C07140=1014.541,221.551,-132.905,168.191,53.842,160.168
C07141=1014.536,221.303,-132.880,168.186,53.852,160.169
C07142=1014.530,221.054,-132.855,168.181,53.862,160.170
C07143=1014.525,220.805,-132.830,168.177,53.871,160.171
C07144=1014.520,220.557,-132.805,168.172,53.881,160.172
C07145=1014.514,220.308,-132.780,168.167,53.891,160.173
C07146=1014.509,220.059,-132.754,168.163,53.900,160.174
C07147=1014.504,219.812,-132.730,168.159,53.910,160.176
C07148=1014.499,219.565,-132.705,168.154,53.919,160.177
C07149=1014.494,219.318,-132.680,168.149,53.929,160.178
C07150=1014.489,219.071,-132.655,168.144,53.939,160.179
C07151=1014.484,218.824,-132.630,168.140,53.948,160.180
C07152=1014.478,218.577,-132.606,168.136,53.959,160.181
C07153=1014.473,218.330,-132.581,168.131,53.969,160.182
C07154=1014.468,218.084,-132.556,168.126,53.978,160.183
C07155=1014.463,217.835,-132.531,168.123,53.988,160.185
C07156=1014.457,217.585,-132.507,168.118,53.997,160.186
C07157=1014.452,217.337,-132.482,168.113,54.008,160.187
C07158=1014.447,217.088,-132.457,168.109,54.018,160.188
C07159=1014.442,216.840,-132.433,168.104,54.027,160.189
C07160=1014.436,216.591,-132.408,168.099,54.038,160.190
C07161=1014.431,216.342,-132.384,168.095,54.048,160.191
C07162=1014.425,216.094,-132.359,168.090,54.058,160.193
C07163=1014.420,215.845,-132.334,168.085,54.068,160.194
C07164=1014.414,215.596,-132.309,168.081,54.078,160.195
C07165=1014.409,215.347,-132.285,168.076,54.088,160.196
C07166=1014.404,215.099,-132.261,168.072,54.099,160.198
C07167=1014.399,214.850,-132.236,168.067,54.108,160.199
C07168=1014.393,214.601,-132.211,168.063,54.119,160.200
C07169=1014.388,214.352,-132.187,168.058,54.129,160.201
C07170=1014.382,214.104,-132.162,168.054,54.139,160.202
C07171=1014.377,213.855,-132.138,168.049,54.149,160.203
C07172=1014.373,213.606,-132.113,168.045,54.159,160.205
C07173=1014.367,213.357,-132.088,168.040,54.169,160.206
C07174=1014.361,213.109,-132.064,168.035,54.180,160.207
C07175=1014.356,212.860,-132.040,168.031,54.190,160.208
C07176=1014.352,212.611,-132.015,168.026,54.200,160.209
C07177=1014.346,212.363,-131.991,168.022,54.211,160.211
C07178=1014.341,212.114,-131.966,168.017,54.220,160.212
C07179=1014.336,211.865,-131.942,168.013,54.231,160.213
C07180=1014.331,211.616,-131.917,168.008,54.241,160.214
C07181=1014.325,211.367,-131.893,168.004,54.251,160.215
C07182=1014.320,211.119,-131.868,168.000,54.262,160.217
C07183=1014.315,210.870,-131.844,167.995,54.272,160.218
C07184=1014.309,210.621,-131.820,167.991,54.282,160.219
C07185=1014.305,210.372,-131.795,167.986,54.293,160.220
C07186=1014.300,210.123,-131.772,167.982,54.303,160.222
C07187=1014.294,209.875,-131.747,167.977,54.313,160.223
C07188=1014.289,209.626,-131.723,167.973,54.324,160.224
C07189=1014.284,209.378,-131.699,167.969,54.334,160.226
C07190=1014.279,209.129,-131.675,167.963,54.345,160.227
C07191=1014.274,208.880,-131.650,167.959,54.355,160.228
C07192=1014.268,208.631,-131.625,167.954,54.365,160.229
C07193=1014.263,208.382,-131.601,167.950,54.376,160.230
C07194=1014.258,208.133,-131.577,167.946,54.386,160.232
C07195=1014.253,207.884,-131.553,167.942,54.397,160.233
C07196=1014.248,207.635,-131.529,167.936,54.408,160.234
C07197=1014.242,207.387,-131.505,167.932,54.418,160.236
C07198=1014.237,207.138,-131.481,167.928,54.429,160.237
C07199=1014.232,206.889,-131.457,167.924,54.440,160.238
C07200=1014.227,206.640,-131.433,167.919,54.450,160.239
C07201=1014.221,206.392,-131.409,167.914,54.461,160.241
C07202=1014.215,206.143,-131.385,167.910,54.472,160.242
C07203=1014.210,205.894,-131.362,167.906,54.482,160.243
C07204=1014.205,205.646,-131.337,167.901,54.493,160.245
C07205=1014.200,205.396,-131.314,167.896,54.504,160.246
C07206=1014.195,205.148,-131.290,167.892,54.514,160.247
C07207=1014.190,204.913,-131.267,167.887,54.524,160.248
C07208=1014.185,204.677,-131.245,167.884,54.534,160.250
C07209=1014.180,204.443,-131.222,167.880,54.545,160.251
C07210=1014.175,204.207,-131.200,167.875,54.555,160.252
C07211=1014.171,203.972,-131.178,167.871,54.565,160.253
C07212=1014.166,203.737,-131.155,167.866,54.575,160.254
C07213=1014.161,203.502,-131.133,167.863,54.585,160.256
C07214=1014.156,203.267,-131.110,167.859,54.596,160.257
C07215=1014.137,202.159,-131.012,167.332,54.506,160.118
C07216=1014.133,201.910,-130.990,167.327,54.518,160.120
C07217=1014.128,201.662,-130.968,167.321,54.530,160.121
C07218=1014.124,201.412,-130.946,167.316,54.542,160.122
C07219=1014.120,201.163,-130.924,167.312,54.554,160.124
C07220=1014.116,200.914,-130.902,167.307,54.566,160.125
C07221=1014.112,200.665,-130.880,167.303,54.577,160.127
C07222=1014.108,200.416,-130.857,167.298,54.589,160.128
C07223=1014.104,200.167,-130.836,167.293,54.600,160.129
C07224=1014.099,199.918,-130.814,167.289,54.612,160.131
C07225=1014.096,199.669,-130.792,167.284,54.625,160.132
C07226=1014.091,199.421,-130.770,167.279,54.636,160.133
C07227=1014.087,199.171,-130.748,167.275,54.648,160.135
C07228=1014.084,198.922,-130.726,167.270,54.660,160.136
C07229=1014.079,198.673,-130.705,167.265,54.672,160.137
C07230=1014.075,198.424,-130.683,167.261,54.684,160.139
C07231=1014.071,198.174,-130.661,167.256,54.696,160.140
C07232=1014.067,197.926,-130.640,167.251,54.708,160.142
C07233=1014.062,197.677,-130.619,167.247,54.720,160.143
C07234=1014.058,197.428,-130.596,167.242,54.732,160.145
C07235=1014.054,197.179,-130.575,167.237,54.744,160.146
C07236=1014.049,196.930,-130.553,167.233,54.756,160.148
C07237=1014.045,196.681,-130.532,167.228,54.768,160.149
C07238=1014.042,196.432,-130.511,167.223,54.780,160.150
C07239=1014.037,196.183,-130.489,167.219,54.792,160.152
C07240=1014.032,195.933,-130.468,167.214,54.804,160.153
C07241=1014.028,195.685,-130.446,167.209,54.816,160.154
C07242=1014.024,195.436,-130.425,167.205,54.828,160.156
C07243=1014.020,195.186,-130.404,167.200,54.840,160.157
C07244=1014.015,194.938,-130.382,167.196,54.852,160.159
C07245=1014.012,194.688,-130.360,167.191,54.863,160.160
C07246=1014.007,194.439,-130.339,167.187,54.876,160.162
C07247=1014.003,194.191,-130.318,167.182,54.888,160.163
C07248=1013.998,193.941,-130.296,167.177,54.900,160.164
C07249=1013.995,193.692,-130.275,167.173,54.912,160.166
C07250=1013.990,193.443,-130.253,167.168,54.924,160.167
C07251=1013.986,193.194,-130.232,167.163,54.936,160.169
C07252=1013.982,192.945,-130.211,167.159,54.947,160.170
C07253=1013.978,192.695,-130.190,167.155,54.960,160.172
C07254=1013.974,192.447,-130.168,167.151,54.971,160.173
C07255=1013.969,192.198,-130.147,167.146,54.983,160.174
C07256=1013.966,191.949,-130.126,167.141,54.995,160.176
C07257=1013.962,191.699,-130.104,167.137,55.008,160.177
C07258=1013.958,191.451,-130.084,167.132,55.019,160.179
C07259=1013.953,191.202,-130.062,167.127,55.031,160.180
C07260=1013.950,190.953,-130.040,167.124,55.043,160.181
C07261=1013.945,190.703,-130.019,167.120,55.055,160.183
C07262=1013.941,190.455,-129.998,167.115,55.067,160.184
C07263=1013.937,190.205,-129.977,167.110,55.079,160.186
C07264=1013.933,189.957,-129.955,167.105,55.091,160.187
C07265=1013.929,189.707,-129.934,167.101,55.103,160.189
C07266=1013.925,189.459,-129.913,167.098,55.115,160.190
C07267=1013.921,189.209,-129.892,167.093,55.127,160.192
C07268=1013.917,188.960,-129.871,167.088,55.138,160.193
C07269=1013.913,188.711,-129.850,167.084,55.151,160.195
C07270=1013.909,188.462,-129.829,167.080,55.162,160.196
C07271=1013.905,188.212,-129.807,167.076,55.174,160.197
C07272=1013.901,187.964,-129.786,167.071,55.186,160.199
C07273=1013.897,187.715,-129.766,167.066,55.198,160.200
C07274=1013.892,187.466,-129.744,167.063,55.210,160.202
C07275=1013.889,187.217,-129.722,167.058,55.222,160.203
C07276=1013.885,186.938,-129.699,167.053,55.235,160.205
C07277=1013.881,186.658,-129.675,167.049,55.249,160.206
C07278=1013.875,186.380,-129.652,167.043,55.262,160.208
C07279=1013.871,186.100,-129.628,167.039,55.275,160.209
C07280=1013.867,185.851,-129.607,167.035,55.287,160.211
C07281=1013.863,185.602,-129.586,167.030,55.299,160.212
C07282=1013.859,185.352,-129.565,167.026,55.311,160.214
C07283=1013.855,185.104,-129.544,167.023,55.323,160.215
C07284=1013.852,184.855,-129.523,167.018,55.335,160.217
C07285=1013.847,184.605,-129.501,167.013,55.347,160.218
C07286=1013.843,184.356,-129.481,167.010,55.358,160.220
C07287=1013.839,184.108,-129.460,167.005,55.370,160.221
C07288=1013.836,183.858,-129.438,167.001,55.382,160.222
C07289=1013.832,183.609,-129.417,166.997,55.393,160.224
C07290=1013.828,183.360,-129.397,166.993,55.406,160.225
C07291=1013.824,183.110,-129.376,166.989,55.418,160.227
C07292=1013.820,182.861,-129.355,166.985,55.430,160.228
C07293=1013.817,182.613,-129.334,166.980,55.441,160.230
C07294=1013.813,182.364,-129.313,166.976,55.453,160.231
C07295=1013.809,182.114,-129.292,166.972,55.465,160.233
C07296=1013.805,181.865,-129.271,166.968,55.476,160.234
C07297=1013.801,181.615,-129.250,166.964,55.488,160.235
C07298=1013.797,181.367,-129.230,166.960,55.501,160.237
C07299=1013.793,181.118,-129.209,166.956,55.512,160.239
C07300=1013.788,180.868,-129.189,166.951,55.524,160.240
C07301=1013.784,180.619,-129.168,166.947,55.537,160.241
C07302=1013.780,180.370,-129.148,166.943,55.549,160.243
C07303=1013.776,180.122,-129.128,166.939,55.561,160.244
C07304=1013.772,179.872,-129.107,166.935,55.573,160.246
C07305=1013.767,179.623,-129.088,166.931,55.585,160.247
C07306=1013.763,179.374,-129.067,166.927,55.598,160.249
C07307=1013.760,179.124,-129.047,166.923,55.609,160.250
C07308=1013.754,178.875,-129.027,166.918,55.621,160.252
C07309=1013.751,178.626,-129.006,166.914,55.634,160.253
C07310=1013.746,178.377,-128.987,166.911,55.645,160.255
C07311=1013.743,178.128,-128.966,166.906,55.657,160.256
C07312=1013.738,177.878,-128.946,166.902,55.670,160.258
C07313=1013.734,177.630,-128.926,166.898,55.682,160.259
C07314=1013.730,177.380,-128.906,166.894,55.694,160.261
C07315=1013.726,177.131,-128.886,166.890,55.706,160.262
C07316=1013.721,176.882,-128.865,166.886,55.718,160.264
C07317=1013.718,176.633,-128.845,166.882,55.730,160.265
C07318=1013.713,176.384,-128.825,166.878,55.743,160.267
C07319=1013.709,176.135,-128.805,166.875,55.754,160.268
C07320=1013.705,175.886,-128.785,166.870,55.766,160.270
C07321=1013.701,175.636,-128.765,166.866,55.778,160.271
C07322=1013.697,175.387,-128.744,166.863,55.790,160.273
C07323=1013.693,175.138,-128.724,166.858,55.802,160.274
C07324=1013.689,174.889,-128.704,166.854,55.814,160.276
C07325=1013.685,174.640,-128.685,166.851,55.827,160.278
C07326=1013.681,174.391,-128.664,166.846,55.839,160.279
C07327=1013.677,174.141,-128.644,166.843,55.850,160.280
C07328=1013.673,173.892,-128.625,166.838,55.862,160.282
C07329=1013.668,173.642,-128.604,166.835,55.875,160.284
C07330=1013.664,173.394,-128.584,166.831,55.887,160.285
C07331=1013.660,173.145,-128.564,166.826,55.899,160.286
C07332=1013.657,172.895,-128.544,166.823,55.910,160.288
C07333=1013.652,172.646,-128.524,166.819,55.923,160.289
C07334=1013.648,172.397,-128.504,166.816,55.935,160.291
C07335=1013.644,172.148,-128.484,166.811,55.947,160.292
C07336=1013.640,171.899,-128.464,166.808,55.958,160.294
C07337=1013.636,171.650,-128.445,166.803,55.970,160.295
C07338=1013.632,171.401,-128.424,166.800,55.983,160.297
C07339=1013.629,171.151,-128.404,166.796,55.995,160.298
C07340=1013.624,170.872,-128.381,166.792,56.007,160.300
C07341=1013.619,170.593,-128.359,166.787,56.021,160.302
C07342=1013.615,170.314,-128.337,166.784,56.034,160.303
C07343=1013.610,170.034,-128.315,166.779,56.048,160.305
C07344=1013.606,169.785,-128.295,166.775,56.060,160.307
C07345=1013.603,169.536,-128.275,166.771,56.072,160.308
C07346=1013.598,169.287,-128.255,166.768,56.083,160.310
C07347=1013.595,169.037,-128.235,166.763,56.095,160.311
C07348=1013.591,168.788,-128.216,166.761,56.108,160.313
C07349=1013.587,168.539,-128.196,166.756,56.120,160.314
C07350=1013.583,168.290,-128.176,166.753,56.131,160.316
C07351=1013.579,168.041,-128.155,166.749,56.143,160.317
C07352=1013.575,167.792,-128.135,166.745,56.155,160.319
C07353=1013.571,167.543,-128.116,166.742,56.167,160.320
C07354=1013.567,167.293,-128.096,166.737,56.179,160.322
C07355=1013.563,167.044,-128.076,166.734,56.190,160.323
C07356=1013.559,166.795,-128.056,166.730,56.202,160.325
C07357=1013.556,166.546,-128.036,166.726,56.214,160.326
C07358=1013.551,166.297,-128.017,166.723,56.227,160.328
C07359=1013.548,166.047,-127.997,166.720,56.238,160.329
C07360=1013.543,165.798,-127.977,166.715,56.250,160.331
C07361=1013.540,165.549,-127.957,166.712,56.262,160.332
C07362=1013.535,165.300,-127.938,166.709,56.274,160.334
C07363=1013.532,165.050,-127.918,166.704,56.286,160.335
C07364=1013.528,164.801,-127.898,166.701,56.297,160.337
C07365=1013.524,164.552,-127.878,166.698,56.309,160.338
C07366=1013.521,164.303,-127.858,166.694,56.321,160.340
C07367=1013.517,164.054,-127.840,166.690,56.333,160.341
C07368=1013.513,163.804,-127.820,166.687,56.345,160.343
C07369=1013.509,163.555,-127.800,166.683,56.356,160.344
C07370=1013.505,163.306,-127.780,166.680,56.368,160.346
C07371=1013.501,163.057,-127.760,166.676,56.380,160.347
C07372=1013.497,162.808,-127.741,166.672,56.392,160.349
C07373=1013.493,162.558,-127.720,166.669,56.403,160.350
C07374=1013.490,162.310,-127.701,166.666,56.415,160.352
C07375=1013.486,162.061,-127.681,166.661,56.427,160.353
C07376=1013.482,161.812,-127.662,166.658,56.439,160.355
C07377=1013.478,161.562,-127.642,166.654,56.450,160.356
C07378=1013.475,161.312,-127.622,166.651,56.462,160.358
C07379=1013.471,161.063,-127.603,166.648,56.473,160.359
C07380=1013.467,160.814,-127.583,166.644,56.485,160.361
C07381=1013.463,160.565,-127.564,166.640,56.497,160.362
C07382=1013.460,160.316,-127.544,166.637,56.509,160.364
C07383=1013.456,160.066,-127.524,166.633,56.521,160.365
C07384=1013.452,159.817,-127.505,166.630,56.532,160.367
C07385=1013.448,159.568,-127.485,166.627,56.544,160.368
C07386=1013.445,159.319,-127.466,166.624,56.556,160.370
C07387=1013.441,159.070,-127.446,166.620,56.567,160.371
C07388=1013.437,158.820,-127.427,166.616,56.579,160.373
C07389=1013.433,158.571,-127.407,166.612,56.591,160.374
C07390=1013.430,158.322,-127.387,166.609,56.603,160.376
C07391=1013.426,158.072,-127.368,166.606,56.614,160.377
C07392=1013.421,157.823,-127.348,166.603,56.626,160.379
C07393=1013.418,157.574,-127.330,166.599,56.638,160.381
C07394=1013.413,157.325,-127.311,166.595,56.650,160.382
C07395=1013.410,157.075,-127.291,166.592,56.662,160.384
C07396=1013.406,156.826,-127.272,166.589,56.673,160.385
C07397=1013.402,156.577,-127.253,166.585,56.685,160.387
C07398=1013.398,156.328,-127.234,166.582,56.697,160.388
C07399=1013.394,156.078,-127.215,166.578,56.709,160.390
C07400=1013.390,155.829,-127.196,166.575,56.721,160.391
C07401=1013.386,155.580,-127.177,166.571,56.733,160.393
C07402=1013.382,155.331,-127.158,166.568,56.744,160.394
C07403=1013.378,155.082,-127.139,166.565,56.756,160.396
C07404=1013.374,154.802,-127.118,166.560,56.769,160.397
C07405=1013.370,154.522,-127.096,166.557,56.783,160.399
C07406=1013.365,154.243,-127.075,166.553,56.796,160.401
C07407=1013.360,153.963,-127.053,166.550,56.809,160.403
C07408=1013.357,153.714,-127.035,166.547,56.821,160.404
C07409=1013.352,153.465,-127.016,166.542,56.833,160.406
C07410=1013.348,153.216,-126.997,166.539,56.845,160.407
C07411=1013.344,152.966,-126.978,166.536,56.857,160.409
C07412=1013.341,152.718,-126.959,166.533,56.868,160.411
C07413=1013.337,152.468,-126.940,166.530,56.880,160.412
C07414=1013.333,152.218,-126.921,166.526,56.891,160.413
C07415=1013.329,151.970,-126.902,166.523,56.903,160.415
C07416=1013.325,151.720,-126.884,166.520,56.915,160.417
C07417=1013.321,151.471,-126.865,166.516,56.927,160.418
C07418=1013.317,151.222,-126.846,166.513,56.938,160.420
C07419=1013.313,150.972,-126.828,166.510,56.950,160.421
C07420=1013.309,150.723,-126.808,166.507,56.962,160.423
C07421=1013.305,150.474,-126.790,166.503,56.974,160.424
C07422=1013.301,150.224,-126.771,166.500,56.986,160.426
C07423=1013.297,149.975,-126.752,166.497,56.998,160.427
C07424=1013.293,149.726,-126.733,166.493,57.009,160.429
C07425=1013.289,149.477,-126.714,166.490,57.021,160.430
C07426=1013.285,149.227,-126.696,166.487,57.033,160.432
C07427=1013.282,148.978,-126.677,166.483,57.044,160.434
C07428=1013.278,148.728,-126.659,166.480,57.056,160.435
C07429=1013.274,148.479,-126.640,166.477,57.068,160.437
C07430=1013.270,148.230,-126.621,166.474,57.079,160.438
C07431=1013.266,147.981,-126.602,166.470,57.091,160.440
C07432=1013.262,147.732,-126.584,166.467,57.103,160.441
C07433=1013.258,147.482,-126.565,166.464,57.115,160.443
C07434=1013.254,147.233,-126.547,166.461,57.126,160.444
C07435=1013.250,146.984,-126.528,166.457,57.138,160.446
C07436=1013.246,146.734,-126.509,166.454,57.149,160.447
C07437=1013.243,146.485,-126.491,166.451,57.161,160.449
C07438=1013.239,146.235,-126.472,166.449,57.173,160.451
C07439=1013.235,145.987,-126.455,166.446,57.184,160.452
C07440=1013.231,145.737,-126.436,166.442,57.196,160.454
C07441=1013.227,145.487,-126.417,166.439,57.207,160.455
C07442=1013.223,145.239,-126.398,166.436,57.219,160.457
C07443=1013.219,144.989,-126.379,166.433,57.231,160.458
C07444=1013.215,144.740,-126.362,166.430,57.242,160.460
C07445=1013.211,144.491,-126.343,166.427,57.254,160.461
C07446=1013.207,144.242,-126.325,166.424,57.266,160.463
C07447=1013.203,143.992,-126.307,166.420,57.278,160.465
C07448=1013.199,143.743,-126.288,166.417,57.290,160.466
C07449=1013.195,143.494,-126.270,166.414,57.301,160.468
C07450=1013.191,143.245,-126.252,166.411,57.313,160.469
C07451=1013.187,142.995,-126.233,166.408,57.325,160.471
C07452=1013.183,142.746,-126.214,166.405,57.336,160.472
C07453=1013.179,142.496,-126.197,166.402,57.347,160.474
C07454=1013.175,142.247,-126.178,166.399,57.359,160.475
C07455=1013.172,141.998,-126.160,166.396,57.371,160.477
C07456=1013.167,141.748,-126.142,166.392,57.382,160.478
C07457=1013.163,141.499,-126.124,166.389,57.394,160.480
C07458=1013.159,141.250,-126.105,166.386,57.406,160.482
C07459=1013.155,141.000,-126.088,166.383,57.417,160.483
C07460=1013.152,140.752,-126.069,166.381,57.428,160.485
C07461=1013.148,140.502,-126.051,166.378,57.440,160.486
C07462=1013.144,140.253,-126.033,166.374,57.452,160.488
C07463=1013.140,140.004,-126.014,166.371,57.463,160.489
C07464=1013.136,139.754,-125.997,166.368,57.475,160.491
C07465=1013.132,139.505,-125.978,166.366,57.486,160.492
C07466=1013.128,139.256,-125.960,166.363,57.498,160.494
C07467=1013.124,139.006,-125.942,166.359,57.509,160.495
C07468=1013.120,138.726,-125.921,166.356,57.522,160.497
C07469=1013.115,138.447,-125.900,166.352,57.535,160.499
C07470=1013.111,138.167,-125.881,166.350,57.548,160.501
C07471=1013.107,137.888,-125.860,166.347,57.561,160.503
C07472=1013.103,137.639,-125.842,166.343,57.572,160.504
C07473=1013.099,137.389,-125.824,166.340,57.584,160.506
C07474=1013.095,137.140,-125.806,166.338,57.595,160.507
C07475=1013.090,136.891,-125.788,166.335,57.607,160.509
C07476=1013.087,136.641,-125.770,166.332,57.619,160.510
C07477=1013.083,136.393,-125.752,166.328,57.630,160.512
C07478=1013.079,136.142,-125.734,166.326,57.641,160.513
C07479=1013.075,135.894,-125.716,166.323,57.653,160.515
C07480=1013.071,135.644,-125.698,166.320,57.665,160.516
C07481=1013.067,135.395,-125.680,166.316,57.676,160.518
C07482=1013.064,135.146,-125.662,166.314,57.687,160.520
C07483=1013.059,134.896,-125.645,166.311,57.698,160.521
C07484=1013.055,134.647,-125.627,166.308,57.710,160.523
C07485=1013.051,134.397,-125.609,166.305,57.721,160.524
C07486=1013.047,134.148,-125.591,166.302,57.733,160.526
C07487=1013.044,133.899,-125.573,166.299,57.744,160.527
C07488=1013.039,133.649,-125.555,166.297,57.756,160.529
C07489=1013.035,133.400,-125.538,166.294,57.767,160.530
C07490=1013.032,133.151,-125.520,166.291,57.779,160.532
C07491=1013.028,132.901,-125.502,166.288,57.790,160.533
C07492=1013.023,132.653,-125.484,166.285,57.802,160.535
C07493=1013.020,132.403,-125.467,166.282,57.813,160.536
C07494=1013.015,132.154,-125.449,166.279,57.824,160.538
C07495=1013.012,131.904,-125.431,166.277,57.836,160.540
C07496=1013.008,131.655,-125.413,166.274,57.847,160.541
C07497=1013.004,131.405,-125.396,166.271,57.859,160.543
C07498=1013.001,131.156,-125.378,166.268,57.870,160.544
C07499=1012.996,130.907,-125.360,166.265,57.881,160.546
C07500=1012.992,130.657,-125.343,166.263,57.893,160.547
C07501=1012.988,130.408,-125.324,166.260,57.903,160.549
C07502=1012.985,130.159,-125.307,166.257,57.915,160.550
C07503=1012.981,129.909,-125.289,166.255,57.926,160.552
C07504=1012.977,129.660,-125.271,166.251,57.937,160.553
C07505=1012.973,129.411,-125.254,166.249,57.948,160.555
C07506=1012.969,129.161,-125.236,166.246,57.960,160.557
C07507=1012.965,128.912,-125.219,166.243,57.972,160.558
C07508=1012.961,128.663,-125.201,166.240,57.982,160.559
C07509=1012.957,128.413,-125.184,166.237,57.994,160.561
C07510=1012.953,128.163,-125.167,166.235,58.005,160.563
C07511=1012.949,127.914,-125.150,166.232,58.017,160.564
C07512=1012.945,127.665,-125.132,166.229,58.028,160.566
C07513=1012.940,127.415,-125.115,166.226,58.039,160.567
C07514=1012.936,127.166,-125.098,166.224,58.051,160.569
C07515=1012.932,126.917,-125.080,166.221,58.062,160.570
C07516=1012.928,126.667,-125.063,166.218,58.073,160.572
C07517=1012.924,126.418,-125.046,166.216,58.085,160.574
C07518=1012.920,126.168,-125.029,166.213,58.096,160.575
C07519=1012.916,125.920,-125.011,166.210,58.107,160.577
C07520=1012.911,125.670,-124.994,166.208,58.119,160.578
C07521=1012.908,125.420,-124.977,166.205,58.130,160.580
C07522=1012.904,125.171,-124.959,166.202,58.141,160.581
C07523=1012.900,124.922,-124.942,166.199,58.152,160.583
C07524=1012.896,124.673,-124.925,166.197,58.164,160.584
C07525=1012.892,124.423,-124.908,166.194,58.175,160.586
C07526=1012.888,124.173,-124.891,166.191,58.186,160.587
C07527=1012.884,123.924,-124.874,166.189,58.197,160.589
C07528=1012.880,123.675,-124.857,166.186,58.208,160.591
C07529=1012.876,123.426,-124.839,166.184,58.220,160.592
C07530=1012.871,123.176,-124.821,166.181,58.231,160.594
C07531=1012.867,122.927,-124.804,166.178,58.242,160.595
C07532=1012.863,122.621,-124.784,166.175,58.255,160.597
C07533=1012.858,122.316,-124.763,166.172,58.269,160.599
C07534=1012.853,122.010,-124.742,166.169,58.282,160.601
C07535=1012.849,121.705,-124.720,166.165,58.296,160.602
C07536=1012.844,121.455,-124.703,166.162,58.307,160.604
C07537=1012.840,121.206,-124.686,166.160,58.318,160.606
C07538=1012.836,120.956,-124.669,166.158,58.330,160.607
C07539=1012.832,120.707,-124.652,166.155,58.341,160.609
C07540=1012.829,120.458,-124.634,166.153,58.352,160.610
C07541=1012.825,120.208,-124.617,166.151,58.363,160.612
C07542=1012.820,119.959,-124.600,166.147,58.374,160.613
C07543=1012.816,119.709,-124.583,166.145,58.385,160.615
C07544=1012.813,119.460,-124.566,166.142,58.395,160.616
C07545=1012.809,119.211,-124.549,166.140,58.406,160.618
C07546=1012.805,118.961,-124.532,166.136,58.417,160.619
C07547=1012.801,118.712,-124.515,166.134,58.428,160.621
C07548=1012.797,118.463,-124.497,166.132,58.439,160.622
C07549=1012.793,118.214,-124.480,166.130,58.450,160.624
C07550=1012.789,117.964,-124.463,166.127,58.461,160.626
C07551=1012.785,117.714,-124.446,166.124,58.472,160.627
C07552=1012.781,117.465,-124.429,166.122,58.483,160.628
C07553=1012.777,117.216,-124.412,166.120,58.494,160.630
C07554=1012.773,116.966,-124.395,166.117,58.504,160.631
C07555=1012.770,116.717,-124.378,166.115,58.515,160.633
C07556=1012.766,116.467,-124.361,166.112,58.526,160.635
C07557=1012.762,116.218,-124.344,166.110,58.537,160.636
C07558=1012.758,115.969,-124.327,166.108,58.548,160.638
C07559=1012.754,115.720,-124.310,166.104,58.558,160.639
C07560=1012.750,115.470,-124.293,166.102,58.569,160.640
C07561=1012.746,115.221,-124.276,166.099,58.580,160.642
C07562=1012.742,114.971,-124.258,166.097,58.591,160.644
C07563=1012.738,114.722,-124.241,166.094,58.601,160.645
C07564=1012.734,114.472,-124.225,166.092,58.612,160.646
C07565=1012.731,114.223,-124.208,166.090,58.623,160.648
C07566=1012.727,113.973,-124.191,166.087,58.633,160.649
C07567=1012.723,113.724,-124.174,166.085,58.644,160.651
C07568=1012.719,113.475,-124.157,166.083,58.655,160.652
C07569=1012.715,113.226,-124.140,166.080,58.665,160.654
C07570=1012.711,112.976,-124.122,166.078,58.676,160.655
C07571=1012.708,112.726,-124.106,166.076,58.687,160.657
C07572=1012.704,112.477,-124.089,166.073,58.697,160.658
C07573=1012.700,112.228,-124.072,166.071,58.708,160.660
C07574=1012.696,111.979,-124.055,166.068,58.719,160.661
C07575=1012.692,111.729,-124.038,166.066,58.729,160.663
C07576=1012.689,111.479,-124.021,166.063,58.740,160.664
C07577=1012.685,111.230,-124.004,166.061,58.751,160.666
C07578=1012.680,110.981,-123.988,166.059,58.762,160.667
C07579=1012.677,110.731,-123.971,166.056,58.772,160.669
C07580=1012.673,110.482,-123.954,166.054,58.783,160.670
C07581=1012.669,110.233,-123.937,166.051,58.794,160.672
C07582=1012.664,109.983,-123.922,166.050,58.803,160.673
C07583=1012.661,109.734,-123.904,166.048,58.814,160.675
C07584=1012.657,109.484,-123.888,166.045,58.825,160.676
C07585=1012.652,109.235,-123.872,166.043,58.836,160.678
C07586=1012.649,108.986,-123.855,166.040,58.846,160.679
C07587=1012.645,108.736,-123.838,166.038,58.857,160.681
C07588=1012.611,121.701,-125.120,166.126,58.488,160.631
C07589=1012.616,121.999,-125.141,166.130,58.476,160.629
C07590=1012.621,122.296,-125.161,166.133,58.462,160.627
C07591=1012.625,122.594,-125.181,166.135,58.450,160.625
C07592=1012.629,122.892,-125.201,166.138,58.436,160.624
C07593=1012.634,123.142,-125.219,166.142,58.425,160.622
C07594=1012.638,123.391,-125.236,166.144,58.414,160.621
C07595=1012.642,123.640,-125.253,166.146,58.403,160.619
C07596=1012.646,123.890,-125.270,166.148,58.392,160.617
C07597=1012.649,124.139,-125.287,166.152,58.381,160.616
C07598=1012.653,124.388,-125.304,166.154,58.370,160.615
C07599=1012.657,124.637,-125.321,166.157,58.359,160.613
C07600=1012.662,124.887,-125.339,166.160,58.348,160.612
C07601=1012.666,125.137,-125.356,166.162,58.337,160.610
C07602=1012.669,125.386,-125.373,166.165,58.326,160.609
C07603=1012.673,125.635,-125.390,166.167,58.314,160.607
C07604=1012.677,125.884,-125.407,166.169,58.303,160.605
C07605=1012.682,126.134,-125.425,166.173,58.292,160.604
C07606=1012.686,126.383,-125.442,166.175,58.281,160.602
C07607=1012.690,126.632,-125.459,166.178,58.270,160.601
C07608=1012.694,126.882,-125.477,166.181,58.259,160.599
C07609=1012.697,127.131,-125.494,166.183,58.247,160.598
C07610=1012.702,127.381,-125.511,166.186,58.236,160.596
C07611=1012.706,127.630,-125.528,166.189,58.225,160.595
C07612=1012.710,127.879,-125.545,166.191,58.214,160.593
C07613=1012.714,128.129,-125.562,166.195,58.202,160.592
C07614=1012.717,128.378,-125.579,166.196,58.191,160.590
C07615=1012.722,128.628,-125.597,166.200,58.180,160.588
C07616=1012.726,128.877,-125.614,166.202,58.169,160.587
C07617=1012.730,129.126,-125.631,166.205,58.157,160.586
C07618=1012.734,129.375,-125.649,166.207,58.146,160.584
C07619=1012.738,129.625,-125.667,166.211,58.135,160.582
C07620=1012.741,129.875,-125.684,166.213,58.124,160.581
C07621=1012.745,130.124,-125.702,166.216,58.112,160.579
C07622=1012.749,130.373,-125.719,166.219,58.102,160.578
C07623=1012.753,130.623,-125.737,166.222,58.090,160.576
C07624=1012.757,130.872,-125.755,166.224,58.079,160.575
C07625=1012.760,131.121,-125.772,166.227,58.067,160.573
C07626=1012.764,131.371,-125.790,166.230,58.057,160.572
C07627=1012.768,131.620,-125.808,166.232,58.045,160.570
C07628=1012.772,131.869,-125.825,166.235,58.034,160.568
C07629=1012.775,132.119,-125.843,166.238,58.023,160.567
C07630=1012.780,132.368,-125.861,166.241,58.012,160.566
C07631=1012.784,132.617,-125.878,166.243,58.000,160.564
C07632=1012.788,132.866,-125.896,166.246,57.989,160.562
C07633=1012.791,133.116,-125.914,166.249,57.978,160.561
C07634=1012.795,133.366,-125.932,166.252,57.966,160.559
C07635=1012.799,133.615,-125.949,166.255,57.955,160.558
C07636=1012.803,133.864,-125.966,166.258,57.944,160.556
C07637=1012.807,134.114,-125.985,166.260,57.932,160.555
C07638=1012.811,134.363,-126.002,166.263,57.921,160.553
C07639=1012.815,134.612,-126.019,166.266,57.909,160.552
C07640=1012.819,134.862,-126.038,166.268,57.898,160.550
C07641=1012.823,135.111,-126.055,166.272,57.887,160.549
C07642=1012.826,135.360,-126.074,166.275,57.875,160.547
C07643=1012.831,135.610,-126.091,166.277,57.864,160.546
C07644=1012.834,135.859,-126.109,166.280,57.852,160.544
C07645=1012.838,136.108,-126.127,166.284,57.841,160.543
C07646=1012.842,136.358,-126.145,166.285,57.829,160.541
C07647=1012.846,136.607,-126.162,166.289,57.818,160.539
C07648=1012.849,136.856,-126.181,166.292,57.807,160.538
C07649=1012.854,137.105,-126.199,166.294,57.795,160.536
C07650=1012.857,137.355,-126.217,166.298,57.784,160.535
C07651=1012.862,137.604,-126.234,166.301,57.772,160.533
C07652=1012.865,137.854,-126.252,166.303,57.761,160.532
C07653=1012.870,138.133,-126.273,166.306,57.748,160.530
C07654=1012.874,138.413,-126.293,166.310,57.735,160.528
C07655=1012.878,138.691,-126.313,166.314,57.723,160.527
C07656=1012.882,138.971,-126.333,166.316,57.710,160.525
C07657=1012.887,139.221,-126.352,166.319,57.698,160.523
C07658=1012.890,139.470,-126.370,166.322,57.687,160.522
C07659=1012.894,139.719,-126.387,166.325,57.675,160.520
C07660=1012.898,139.969,-126.406,166.328,57.664,160.519
C07661=1012.902,140.217,-126.424,166.331,57.652,160.517
C07662=1012.906,140.467,-126.443,166.334,57.641,160.516
C07663=1012.909,140.717,-126.460,166.337,57.629,160.514
C07664=1012.914,140.966,-126.478,166.341,57.618,160.513
C07665=1012.917,141.215,-126.497,166.343,57.606,160.511
C07666=1012.921,141.464,-126.515,166.346,57.594,160.509
C07667=1012.925,141.714,-126.533,166.349,57.583,160.508
C07668=1012.929,141.963,-126.551,166.352,57.571,160.506
C07669=1012.933,142.212,-126.570,166.356,57.560,160.505
C07670=1012.937,142.461,-126.588,166.359,57.548,160.503
C07671=1012.941,142.711,-126.606,166.361,57.537,160.501
C07672=1012.944,142.960,-126.624,166.364,57.526,160.500
C07673=1012.949,143.210,-126.642,166.367,57.514,160.498
C07674=1012.952,143.459,-126.661,166.370,57.502,160.497
C07675=1012.956,143.708,-126.679,166.374,57.491,160.496
C07676=1012.960,143.958,-126.696,166.377,57.479,160.494
C07677=1012.964,144.206,-126.715,166.380,57.467,160.492
C07678=1012.968,144.456,-126.734,166.383,57.455,160.491
C07679=1012.972,144.705,-126.751,166.386,57.444,160.489
C07680=1012.976,144.954,-126.770,166.389,57.432,160.488
C07681=1012.979,145.203,-126.789,166.392,57.420,160.486
C07682=1012.984,145.453,-126.807,166.395,57.409,160.485
C07683=1012.987,145.702,-126.824,166.398,57.397,160.483
C07684=1012.991,145.952,-126.843,166.401,57.385,160.481
C07685=1012.995,146.202,-126.862,166.404,57.374,160.480
C07686=1012.999,146.451,-126.880,166.407,57.362,160.478
C07687=1013.003,146.700,-126.899,166.410,57.351,160.477
C07688=1013.006,146.949,-126.917,166.414,57.339,160.475
C07689=1013.010,147.199,-126.936,166.417,57.327,160.474
C07690=1013.015,147.448,-126.954,166.420,57.316,160.472
C07691=1013.019,147.697,-126.973,166.423,57.304,160.471
C07692=1013.022,147.946,-126.991,166.426,57.292,160.469
C07693=1013.026,148.196,-127.010,166.430,57.281,160.468
C07694=1013.030,148.444,-127.029,166.433,57.269,160.466
C07695=1013.034,148.694,-127.048,166.436,57.257,160.464
C07696=1013.038,148.943,-127.066,166.439,57.245,160.463
C07697=1013.041,149.192,-127.085,166.443,57.234,160.462
C07698=1013.045,149.442,-127.104,166.446,57.222,160.460
C07699=1013.049,149.691,-127.122,166.449,57.210,160.458
C07700=1013.053,149.941,-127.141,166.452,57.198,160.457
C07701=1013.056,150.190,-127.159,166.455,57.187,160.455
C07702=1013.060,150.439,-127.178,166.459,57.176,160.454
C07703=1013.065,150.688,-127.197,166.462,57.164,160.452
C07704=1013.069,150.937,-127.215,166.465,57.152,160.451
C07705=1013.073,151.187,-127.234,166.468,57.140,160.449
C07706=1013.076,151.436,-127.252,166.471,57.128,160.447
C07707=1013.081,151.685,-127.271,166.474,57.116,160.446
C07708=1013.085,151.935,-127.290,166.477,57.104,160.444
C07709=1013.088,152.184,-127.308,166.482,57.093,160.443
C07710=1013.092,152.433,-127.328,166.485,57.081,160.441
C07711=1013.096,152.683,-127.346,166.488,57.069,160.440
C07712=1013.100,152.932,-127.365,166.491,57.057,160.438
C07713=1013.104,153.181,-127.384,166.494,57.046,160.437
C07714=1013.107,153.430,-127.403,166.497,57.034,160.435
C07715=1013.111,153.680,-127.422,166.501,57.022,160.434
C07716=1013.115,153.929,-127.441,166.504,57.011,160.432
C07717=1013.120,154.208,-127.462,166.507,56.997,160.430
C07718=1013.124,154.487,-127.483,166.512,56.984,160.429
C07719=1013.128,154.767,-127.505,166.516,56.971,160.427
C07720=1013.133,155.047,-127.526,166.519,56.958,160.425
C07721=1013.137,155.295,-127.545,166.522,56.946,160.424
C07722=1013.141,155.545,-127.563,166.527,56.934,160.422
C07723=1013.144,155.795,-127.583,166.530,56.922,160.421
C07724=1013.148,156.043,-127.602,166.533,56.910,160.419
C07725=1013.152,156.293,-127.621,166.536,56.899,160.418
C07726=1013.156,156.542,-127.639,166.539,56.887,160.416
C07727=1013.160,156.791,-127.659,166.543,56.875,160.415
C07728=1013.163,157.040,-127.677,166.547,56.863,160.413
C07729=1013.168,157.289,-127.697,166.550,56.851,160.411
C07730=1013.172,157.539,-127.715,166.553,56.839,160.410
C07731=1013.175,157.788,-127.734,166.557,56.827,160.408
C07732=1013.180,158.037,-127.753,166.560,56.815,160.407
C07733=1013.183,158.287,-127.773,166.563,56.803,160.405
C07734=1013.187,158.536,-127.792,166.567,56.792,160.404
C07735=1013.191,158.785,-127.812,166.570,56.780,160.402
C07736=1013.194,159.035,-127.831,166.573,56.768,160.400
C07737=1013.198,159.284,-127.851,166.577,56.757,160.399
C07738=1013.202,159.533,-127.871,166.581,56.745,160.398
C07739=1013.206,159.783,-127.890,166.584,56.733,160.396
C07740=1013.209,160.031,-127.909,166.588,56.721,160.395
C07741=1013.212,160.281,-127.929,166.591,56.710,160.393
C07742=1013.217,160.530,-127.949,166.594,56.698,160.391
C07743=1013.220,160.780,-127.968,166.597,56.686,160.390
C07744=1013.224,161.028,-127.987,166.601,56.674,160.389
C07745=1013.227,161.277,-128.007,166.605,56.662,160.387
C07746=1013.232,161.526,-128.027,166.608,56.651,160.386
C07747=1013.235,161.776,-128.046,166.612,56.639,160.384
C07748=1013.239,162.026,-128.066,166.615,56.628,160.383
C07749=1013.242,162.274,-128.085,166.619,56.615,160.381
C07750=1013.246,162.523,-128.105,166.622,56.604,160.380
C07751=1013.250,162.772,-128.125,166.626,56.592,160.378
C07752=1013.254,163.022,-128.144,166.629,56.580,160.376
C07753=1013.258,163.271,-128.164,166.633,56.568,160.375
C07754=1013.261,163.520,-128.183,166.637,56.556,160.373
C07755=1013.265,163.769,-128.203,166.640,56.545,160.372
C07756=1013.269,164.019,-128.223,166.644,56.533,160.371
C07757=1013.272,164.268,-128.243,166.647,56.521,160.369
C07758=1013.277,164.517,-128.262,166.651,56.509,160.367
C07759=1013.280,164.767,-128.282,166.655,56.497,160.366
C07760=1013.283,165.016,-128.301,166.658,56.485,160.364
C07761=1013.287,165.265,-128.321,166.662,56.473,160.363
C07762=1013.291,165.514,-128.341,166.666,56.461,160.361
C07763=1013.295,165.763,-128.360,166.669,56.450,160.360
C07764=1013.299,166.012,-128.381,166.672,56.438,160.358
C07765=1013.303,166.261,-128.400,166.677,56.426,160.357
C07766=1013.307,166.511,-128.420,166.680,56.414,160.355
C07767=1013.311,166.760,-128.440,166.683,56.402,160.354
C07768=1013.315,167.009,-128.460,166.687,56.390,160.352
C07769=1013.318,167.258,-128.479,166.690,56.378,160.351
C07770=1013.322,167.507,-128.498,166.695,56.366,160.349
C07771=1013.326,167.757,-128.518,166.698,56.354,160.348
C07772=1013.329,168.006,-128.538,166.701,56.342,160.346
C07773=1013.334,168.255,-128.558,166.706,56.330,160.345
C07774=1013.337,168.505,-128.578,166.709,56.319,160.343
C07775=1013.342,168.754,-128.597,166.714,56.307,160.342
C07776=1013.345,169.003,-128.617,166.716,56.294,160.340
C07777=1013.349,169.252,-128.637,166.721,56.282,160.339
C07778=1013.353,169.501,-128.657,166.724,56.270,160.337
C07779=1013.357,169.751,-128.677,166.728,56.258,160.336
C07780=1013.361,170.000,-128.696,166.732,56.247,160.334
C07781=1013.366,170.278,-128.719,166.736,56.233,160.332
C07782=1013.370,170.557,-128.741,166.740,56.220,160.331
C07783=1013.374,170.837,-128.764,166.744,56.206,160.329
C07784=1013.379,171.116,-128.786,166.749,56.193,160.327
C07785=1013.383,171.365,-128.806,166.752,56.180,160.326
C07786=1013.386,171.615,-128.826,166.756,56.168,160.324
C07787=1013.391,171.864,-128.845,166.760,56.157,160.323
C07788=1013.394,172.113,-128.865,166.764,56.145,160.321
C07789=1013.398,172.362,-128.885,166.768,56.133,160.320
C07790=1013.402,172.611,-128.905,166.772,56.120,160.318
C07791=1013.406,172.861,-128.925,166.776,56.108,160.317
C07792=1013.411,173.109,-128.945,166.779,56.096,160.315
C07793=1013.414,173.359,-128.965,166.784,56.084,160.314
C07794=1013.418,173.608,-128.985,166.787,56.072,160.312
C07795=1013.422,173.857,-129.005,166.791,56.060,160.311
C07796=1013.426,174.106,-129.025,166.796,56.048,160.309
C07797=1013.430,174.355,-129.044,166.798,56.036,160.307
C07798=1013.434,174.604,-129.065,166.803,56.024,160.306
C07799=1013.438,174.853,-129.085,166.807,56.011,160.305
C07800=1013.443,175.103,-129.105,166.811,56.000,160.303
C07801=1013.446,175.352,-129.125,166.815,55.987,160.302
C07802=1013.451,175.602,-129.144,166.818,55.976,160.300
C07803=1013.455,175.850,-129.165,166.823,55.963,160.299
C07804=1013.458,176.100,-129.185,166.826,55.951,160.297
C07805=1013.462,176.349,-129.205,166.831,55.939,160.296
C07806=1013.466,176.598,-129.225,166.834,55.927,160.294
C07807=1013.471,176.846,-129.245,166.838,55.914,160.292
C07808=1013.474,177.096,-129.265,166.843,55.902,160.291
C07809=1013.479,177.346,-129.285,166.846,55.891,160.290
C07810=1013.483,177.595,-129.305,166.850,55.878,160.288
C07811=1013.487,177.844,-129.326,166.855,55.866,160.287
C07812=1013.491,178.093,-129.345,166.859,55.853,160.285
C07813=1013.495,178.342,-129.365,166.862,55.842,160.283
C07814=1013.499,178.590,-129.385,166.867,55.830,160.282
C07815=1013.504,178.840,-129.406,166.871,55.817,160.280
C07816=1013.507,179.090,-129.426,166.875,55.805,160.279
C07817=1013.512,179.338,-129.446,166.879,55.793,160.277
C07818=1013.516,179.588,-129.466,166.883,55.781,160.276
C07819=1013.520,179.837,-129.486,166.887,55.769,160.274
C07820=1013.524,180.086,-129.507,166.891,55.756,160.273
C07821=1013.528,180.335,-129.527,166.896,55.744,160.272
C07822=1013.532,180.584,-129.546,166.899,55.732,160.270
C07823=1013.536,180.833,-129.567,166.903,55.720,160.268
C07824=1013.541,181.082,-129.587,166.908,55.708,160.267
C07825=1013.545,181.332,-129.608,166.912,55.695,160.265
C07826=1013.549,181.581,-129.628,166.916,55.683,160.264
C07827=1013.552,181.830,-129.649,166.920,55.672,160.262
C07828=1013.556,182.080,-129.670,166.924,55.660,160.261
C07829=1013.560,182.329,-129.690,166.928,55.647,160.259
C07830=1013.564,182.578,-129.711,166.932,55.635,160.258
C07831=1013.567,182.827,-129.733,166.936,55.623,160.257
C07832=1013.572,183.076,-129.754,166.941,55.612,160.255
C07833=1013.575,183.325,-129.774,166.944,55.600,160.254
C07834=1013.579,183.574,-129.794,166.949,55.588,160.252
C07835=1013.582,183.823,-129.816,166.953,55.575,160.251
C07836=1013.587,184.073,-129.837,166.957,55.564,160.249
C07837=1013.591,184.321,-129.858,166.961,55.552,160.248
C07838=1013.595,184.570,-129.879,166.966,55.540,160.247
C07839=1013.598,184.819,-129.900,166.969,55.528,160.245
C07840=1013.602,185.069,-129.920,166.973,55.516,160.243
C07841=1013.606,185.318,-129.941,166.978,55.504,160.242
C07842=1013.610,185.567,-129.962,166.983,55.492,160.241
C07843=1013.614,185.816,-129.984,166.986,55.480,160.239
C07844=1013.618,186.065,-130.004,166.990,55.468,160.238
C07845=1013.622,186.344,-130.028,166.995,55.455,160.236
C07846=1013.626,186.624,-130.052,167.000,55.441,160.234
C07847=1013.631,186.903,-130.075,167.005,55.428,160.233
C07848=1013.635,187.182,-130.099,167.010,55.414,160.231
C07849=1013.639,187.431,-130.120,167.014,55.402,160.230
C07850=1013.643,187.680,-130.140,167.019,55.390,160.228
C07851=1013.647,187.929,-130.162,167.022,55.378,160.227
C07852=1013.651,188.178,-130.183,167.027,55.366,160.225
C07853=1013.654,188.427,-130.204,167.031,55.354,160.224
C07854=1013.659,188.676,-130.225,167.035,55.342,160.222
C07855=1013.663,188.925,-130.246,167.040,55.330,160.221
C07856=1013.667,189.175,-130.267,167.045,55.318,160.220
C07857=1013.671,189.423,-130.288,167.049,55.306,160.218
C07858=1013.674,189.672,-130.309,167.052,55.294,160.217
C07859=1013.679,189.921,-130.331,167.057,55.282,160.215
C07860=1013.682,190.170,-130.352,167.062,55.270,160.214
C07861=1013.687,190.419,-130.373,167.066,55.258,160.212
C07862=1013.691,190.668,-130.394,167.071,55.246,160.211
C07863=1013.695,190.918,-130.416,167.075,55.234,160.210
C07864=1013.699,191.167,-130.437,167.079,55.221,160.208
C07865=1013.703,191.415,-130.457,167.084,55.209,160.207
C07866=1013.707,191.665,-130.479,167.089,55.197,160.205
C07867=1013.710,191.914,-130.500,167.093,55.185,160.204
C07868=1013.715,192.163,-130.521,167.098,55.173,160.202
C07869=1013.719,192.411,-130.543,167.102,55.161,160.201
C07870=1013.723,192.661,-130.564,167.105,55.149,160.199
C07871=1013.727,192.910,-130.585,167.110,55.137,160.198
C07872=1013.731,193.159,-130.606,167.115,55.125,160.196
C07873=1013.735,193.408,-130.627,167.119,55.113,160.195
C07874=1013.739,193.657,-130.650,167.124,55.101,160.194
C07875=1013.743,193.906,-130.670,167.128,55.089,160.192
C07876=1013.748,194.155,-130.691,167.133,55.077,160.191
C07877=1013.752,194.404,-130.712,167.137,55.065,160.189
C07878=1013.755,194.654,-130.734,167.142,55.053,160.188
C07879=1013.760,194.903,-130.756,167.146,55.040,160.186
C07880=1013.764,195.151,-130.777,167.152,55.028,160.185
C07881=1013.769,195.401,-130.798,167.156,55.016,160.183
C07882=1013.772,195.650,-130.819,167.161,55.004,160.182
C07883=1013.777,195.899,-130.841,167.166,54.992,160.181
C07884=1013.780,196.147,-130.862,167.170,54.979,160.179
C07885=1013.784,196.397,-130.884,167.175,54.968,160.178
C07886=1013.789,196.646,-130.905,167.179,54.955,160.176
C07887=1013.793,196.895,-130.926,167.184,54.943,160.175
C07888=1013.798,197.144,-130.947,167.188,54.931,160.174
C07889=1013.802,197.393,-130.970,167.192,54.919,160.172
C07890=1013.806,197.642,-130.991,167.197,54.907,160.171
C07891=1013.810,197.891,-131.012,167.201,54.895,160.169
C07892=1013.814,198.140,-131.033,167.207,54.882,160.168
C07893=1013.818,198.389,-131.055,167.212,54.871,160.166
C07894=1013.823,198.638,-131.077,167.216,54.858,160.165
C07895=1013.827,198.887,-131.098,167.221,54.846,160.164
C07896=1013.831,199.136,-131.120,167.226,54.835,160.162
C07897=1013.835,199.386,-131.142,167.230,54.822,160.161
C07898=1013.839,199.634,-131.163,167.235,54.810,160.159
C07899=1013.843,199.884,-131.185,167.240,54.799,160.158
C07900=1013.847,200.133,-131.208,167.244,54.786,160.156
C07901=1013.851,200.381,-131.229,167.249,54.774,160.155
C07902=1013.855,200.631,-131.251,167.254,54.763,160.154
C07903=1013.859,200.880,-131.273,167.258,54.751,160.152
C07904=1013.864,201.129,-131.295,167.263,54.738,160.151
C07905=1013.867,201.378,-131.316,167.268,54.726,160.150
C07906=1013.871,201.627,-131.339,167.273,54.714,160.148
C07907=1013.876,201.876,-131.361,167.278,54.703,160.147
C07908=1013.879,202.124,-131.383,167.282,54.690,160.145
C07909=1013.897,203.217,-131.479,167.813,54.786,160.288
C07910=1013.902,203.455,-131.502,167.817,54.776,160.286
C07911=1013.907,203.693,-131.524,167.821,54.765,160.285
C07912=1013.912,203.931,-131.547,167.825,54.755,160.284
C07913=1013.917,204.169,-131.570,167.830,54.745,160.283
C07914=1013.922,204.408,-131.592,167.834,54.734,160.281
C07915=1013.927,204.646,-131.616,167.838,54.723,160.280
C07916=1013.932,204.884,-131.638,167.842,54.713,160.279
C07917=1013.937,205.122,-131.660,167.847,54.703,160.278
C07918=1013.942,205.370,-131.685,167.851,54.692,160.276
C07919=1013.947,205.620,-131.708,167.856,54.681,160.275
C07920=1013.952,205.868,-131.732,167.860,54.670,160.273
C07921=1013.957,206.117,-131.756,167.864,54.659,160.272
C07922=1013.963,206.366,-131.780,167.869,54.648,160.271
C07923=1013.968,206.615,-131.804,167.874,54.638,160.270
C07924=1013.973,206.864,-131.828,167.878,54.627,160.268
C07925=1013.978,207.112,-131.852,167.883,54.616,160.267
C07926=1013.983,207.362,-131.876,167.887,54.606,160.266
C07927=1013.989,207.610,-131.900,167.891,54.595,160.264
C07928=1013.994,207.859,-131.924,167.897,54.584,160.263
C07929=1013.999,208.108,-131.948,167.901,54.573,160.262
C07930=1014.004,208.357,-131.972,167.905,54.563,160.261
C07931=1014.009,208.605,-131.996,167.909,54.552,160.259
C07932=1014.014,208.854,-132.020,167.914,54.541,160.258
C07933=1014.020,209.103,-132.044,167.919,54.531,160.257
C07934=1014.025,209.352,-132.068,167.923,54.520,160.255
C07935=1014.030,209.600,-132.093,167.927,54.510,160.254
C07936=1014.035,209.849,-132.116,167.932,54.499,160.253
C07937=1014.041,210.098,-132.140,167.937,54.489,160.252
C07938=1014.045,210.347,-132.165,167.941,54.478,160.250
C07939=1014.050,210.595,-132.189,167.945,54.468,160.249
C07940=1014.056,210.844,-132.214,167.950,54.457,160.248
C07941=1014.061,211.093,-132.238,167.954,54.447,160.247
C07942=1014.066,211.342,-132.262,167.960,54.436,160.246
C07943=1014.071,211.591,-132.286,167.964,54.426,160.244
C07944=1014.076,211.839,-132.311,167.968,54.415,160.243
C07945=1014.081,212.088,-132.335,167.973,54.405,160.242
C07946=1014.087,212.337,-132.359,167.977,54.395,160.241
C07947=1014.091,212.585,-132.384,167.981,54.384,160.239
C07948=1014.097,212.835,-132.409,167.986,54.374,160.238
C07949=1014.102,213.083,-132.433,167.991,54.364,160.237
C07950=1014.108,213.332,-132.457,167.996,54.353,160.236
C07951=1014.113,213.580,-132.481,168.000,54.343,160.235
C07952=1014.117,213.829,-132.506,168.005,54.333,160.233
C07953=1014.123,214.078,-132.531,168.009,54.322,160.232
C07954=1014.128,214.327,-132.555,168.014,54.312,160.231
C07955=1014.133,214.575,-132.579,168.018,54.302,160.230
C07956=1014.139,214.825,-132.604,168.023,54.292,160.228
C07957=1014.144,215.073,-132.629,168.027,54.281,160.227
C07958=1014.149,215.322,-132.653,168.032,54.270,160.226
C07959=1014.154,215.570,-132.677,168.037,54.261,160.225
C07960=1014.160,215.819,-132.701,168.041,54.250,160.224
C07961=1014.165,216.069,-132.726,168.046,54.240,160.223
C07962=1014.170,216.317,-132.751,168.050,54.230,160.221
C07963=1014.175,216.566,-132.775,168.055,54.220,160.220
C07964=1014.181,216.814,-132.800,168.059,54.210,160.219
C07965=1014.186,217.063,-132.825,168.064,54.200,160.218
C07966=1014.192,217.312,-132.849,168.069,54.189,160.216
C07967=1014.197,217.561,-132.874,168.073,54.179,160.215
C07968=1014.202,217.809,-132.898,168.078,54.169,160.214
C07969=1014.207,218.057,-132.924,168.082,54.159,160.213
C07970=1014.212,218.306,-132.948,168.087,54.149,160.212
C07971=1014.218,218.554,-132.973,168.092,54.140,160.211
C07972=1014.223,218.802,-132.998,168.096,54.129,160.210
C07973=1014.227,219.050,-133.022,168.101,54.119,160.208
C07974=1014.233,219.298,-133.047,168.106,54.109,160.207
C07975=1014.238,219.546,-133.073,168.111,54.100,160.206
C07976=1014.243,219.795,-133.097,168.114,54.090,160.205
C07977=1014.249,220.043,-133.122,168.119,54.080,160.204
C07978=1014.253,220.292,-133.147,168.124,54.070,160.203
C07979=1014.259,220.540,-133.172,168.128,54.060,160.202
C07980=1014.264,220.789,-133.197,168.133,54.050,160.201
C07981=1014.270,221.037,-133.222,168.138,54.041,160.200
C07982=1014.274,221.286,-133.247,168.142,54.030,160.198
C07983=1014.279,221.536,-133.272,168.147,54.020,160.197
C07984=1014.285,221.784,-133.297,168.152,54.011,160.196
C07985=1014.290,222.033,-133.322,168.156,54.001,160.195
C07986=1014.296,222.281,-133.347,168.161,53.992,160.194
C07987=1014.300,222.530,-133.372,168.165,53.982,160.193
C07988=1014.306,222.778,-133.397,168.170,53.972,160.192
C07989=1014.311,223.028,-133.422,168.175,53.962,160.191
C07990=1014.317,223.276,-133.447,168.180,53.953,160.190
C07991=1014.322,223.525,-133.473,168.184,53.942,160.188
C07992=1014.328,223.773,-133.497,168.188,53.933,160.187
C07993=1014.332,224.022,-133.523,168.193,53.923,160.186
C07994=1014.338,224.271,-133.548,168.198,53.913,160.185
C07995=1014.343,224.519,-133.573,168.203,53.903,160.184
C07996=1014.349,224.769,-133.598,168.207,53.894,160.183
C07997=1014.354,225.017,-133.623,168.212,53.884,160.182
C07998=1014.359,225.266,-133.649,168.216,53.875,160.180
C07999=1014.365,225.514,-133.674,168.221,53.865,160.179
C08000=1014.370,225.763,-133.699,168.226,53.856,160.179
C08001=1014.376,226.011,-133.724,168.231,53.846,160.178
C08002=1014.380,226.260,-133.749,168.235,53.837,160.176
C08003=1014.386,226.509,-133.775,168.240,53.827,160.175
C08004=1014.391,226.757,-133.800,168.245,53.817,160.174
C08005=1014.397,227.006,-133.826,168.250,53.808,160.173
C08006=1014.402,227.254,-133.852,168.254,53.799,160.172
C08007=1014.407,227.504,-133.877,168.259,53.789,160.171
C08008=1014.412,227.752,-133.902,168.264,53.779,160.170
C08009=1014.418,228.001,-133.928,168.268,53.770,160.169
C08010=1014.423,228.249,-133.953,168.273,53.761,160.168
C08011=1014.428,228.498,-133.979,168.278,53.751,160.167
C08012=1014.433,228.747,-134.005,168.282,53.742,160.166
C08013=1014.439,228.995,-134.031,168.287,53.733,160.165
C08014=1014.444,229.243,-134.056,168.292,53.723,160.164
C08015=1014.449,229.493,-134.081,168.296,53.714,160.163
C08016=1014.454,229.741,-134.107,168.301,53.705,160.162
C08017=1014.460,229.990,-134.133,168.306,53.695,160.161
C08018=1014.465,230.238,-134.159,168.310,53.687,160.160
C08019=1014.470,230.487,-134.185,168.315,53.677,160.159
C08020=1014.476,230.736,-134.211,168.320,53.667,160.158
C08021=1014.481,230.984,-134.236,168.324,53.659,160.157
C08022=1014.486,231.233,-134.262,168.329,53.649,160.156
C08023=1014.491,231.481,-134.288,168.334,53.640,160.155
C08024=1014.497,231.730,-134.314,168.339,53.631,160.154
C08025=1014.502,231.978,-134.339,168.343,53.622,160.153
C08026=1014.508,232.227,-134.365,168.348,53.613,160.152
C08027=1014.513,232.476,-134.390,168.353,53.603,160.151
C08028=1014.518,232.725,-134.416,168.358,53.595,160.150
C08029=1014.524,232.973,-134.443,168.362,53.585,160.149
C08030=1014.528,233.218,-134.468,168.367,53.577,160.148
C08031=1014.534,233.461,-134.493,168.372,53.568,160.147
C08032=1014.539,233.705,-134.519,168.377,53.559,160.146
C08033=1014.545,233.948,-134.544,168.380,53.550,160.145
C08034=1014.550,234.194,-134.570,168.386,53.541,160.144
C08035=1014.555,234.437,-134.595,168.390,53.532,160.143
C08036=1014.561,234.681,-134.621,168.396,53.523,160.142
C08037=1014.566,234.925,-134.646,168.400,53.514,160.141
C08038=1014.571,235.174,-134.672,168.404,53.505,160.140
C08039=1014.576,235.422,-134.698,168.409,53.496,160.139
C08040=1014.582,235.671,-134.724,168.414,53.488,160.138
C08041=1014.588,235.919,-134.750,168.419,53.478,160.137
C08042=1014.592,236.167,-134.776,168.423,53.469,160.136
C08043=1014.598,236.416,-134.802,168.428,53.460,160.136
C08044=1014.604,236.665,-134.828,168.433,53.452,160.135
C08045=1014.609,236.914,-134.854,168.438,53.442,160.134
C08046=1014.614,237.161,-134.881,168.442,53.434,160.133
C08047=1014.620,237.410,-134.907,168.447,53.425,160.132
C08048=1014.625,237.659,-134.933,168.452,53.416,160.131
C08049=1014.631,237.908,-134.959,168.457,53.407,160.130
C08050=1014.636,238.156,-134.985,168.462,53.399,160.129
C08051=1014.642,238.404,-135.011,168.467,53.390,160.128
C08052=1014.646,238.654,-135.038,168.471,53.380,160.127
C08053=1014.652,238.902,-135.065,168.476,53.371,160.126
C08054=1014.657,239.150,-135.090,168.481,53.363,160.125
C08055=1014.663,239.399,-135.117,168.485,53.354,160.124
C08056=1014.668,239.647,-135.144,168.491,53.346,160.124
C08057=1014.673,239.896,-135.170,168.496,53.337,160.123
C08058=1014.679,240.145,-135.197,168.500,53.329,160.122
C08059=1014.684,240.393,-135.224,168.505,53.320,160.121
C08060=1014.689,240.642,-135.249,168.510,53.311,160.120
C08061=1014.695,240.890,-135.276,168.515,53.303,160.119
C08062=1014.701,241.138,-135.303,168.520,53.294,160.118
C08063=1014.705,241.388,-135.329,168.524,53.285,160.117
C08064=1014.711,241.636,-135.356,168.529,53.276,160.116
C08065=1014.717,241.884,-135.383,168.534,53.268,160.115
C08066=1014.721,242.132,-135.409,168.539,53.260,160.115
C08067=1014.727,242.381,-135.435,168.544,53.251,160.114
C08068=1014.733,242.630,-135.462,168.549,53.243,160.113
C08069=1014.738,242.878,-135.489,168.553,53.234,160.112
C08070=1014.743,243.127,-135.516,168.558,53.226,160.111
C08071=1014.748,243.375,-135.543,168.563,53.217,160.110
C08072=1014.754,243.624,-135.570,168.568,53.209,160.110
C08073=1014.759,243.872,-135.597,168.573,53.201,160.109
C08074=1014.764,244.120,-135.624,168.577,53.192,160.108
C08075=1014.769,244.369,-135.651,168.583,53.184,160.107
C08076=1014.774,244.617,-135.678,168.587,53.176,160.106
C08077=1014.780,244.866,-135.704,168.592,53.167,160.105
C08078=1014.785,245.114,-135.732,168.597,53.159,160.105
C08079=1014.791,245.363,-135.758,168.601,53.151,160.104
C08080=1014.796,245.611,-135.786,168.607,53.143,160.103
C08081=1014.801,245.860,-135.813,168.612,53.134,160.102
C08082=1014.807,246.109,-135.839,168.617,53.126,160.101
C08083=1014.812,246.357,-135.867,168.621,53.118,160.100
C08084=1014.818,246.606,-135.893,168.626,53.110,160.100
C08085=1014.823,246.854,-135.921,168.631,53.101,160.099
C08086=1014.828,247.103,-135.948,168.636,53.093,160.098
C08087=1014.834,247.351,-135.974,168.641,53.085,160.097
C08088=1014.839,247.599,-136.002,168.646,53.077,160.097
C08089=1014.845,247.848,-136.029,168.650,53.068,160.096
C08090=1014.850,248.089,-136.055,168.655,53.060,160.095
C08091=1014.855,248.329,-136.082,168.660,53.053,160.094
C08092=1014.860,248.570,-136.108,168.665,53.045,160.093
C08093=1014.866,248.810,-136.134,168.670,53.037,160.093
C08094=1014.870,249.051,-136.161,168.675,53.029,160.092
C08095=1014.876,249.291,-136.187,168.680,53.021,160.091
C08096=1014.881,249.532,-136.213,168.684,53.013,160.090
C08097=1014.886,249.772,-136.240,168.689,53.005,160.090
C08098=1014.891,250.021,-136.267,168.694,52.997,160.089
C08099=1014.897,250.269,-136.294,168.699,52.989,160.088
C08100=1014.903,250.517,-136.322,168.703,52.981,160.087
C08101=1014.908,250.766,-136.348,168.708,52.973,160.086
C08102=1014.914,251.015,-136.376,168.713,52.965,160.086
C08103=1014.919,251.264,-136.403,168.719,52.957,160.085
C08104=1014.925,251.511,-136.430,168.723,52.949,160.084
C08105=1014.930,251.760,-136.458,168.728,52.941,160.083
C08106=1014.936,252.008,-136.484,168.733,52.933,160.083
C08107=1014.941,252.256,-136.512,168.738,52.925,160.082
C08108=1014.947,252.506,-136.540,168.743,52.917,160.081
C08109=1014.953,252.753,-136.567,168.748,52.909,160.080
C08110=1014.958,253.002,-136.594,168.754,52.901,160.080
C08111=1014.964,253.251,-136.621,168.759,52.893,160.079
C08112=1014.969,253.499,-136.649,168.763,52.885,160.078
C08113=1014.975,253.748,-136.677,168.768,52.878,160.078
C08114=1014.981,253.996,-136.704,168.773,52.870,160.077
C08115=1014.986,254.244,-136.731,168.778,52.861,160.076
C08116=1014.992,254.492,-136.759,168.783,52.854,160.075
C08117=1014.998,254.741,-136.786,168.788,52.846,160.074
C08118=1015.003,254.990,-136.814,168.793,52.838,160.074
C08119=1015.009,255.238,-136.841,168.799,52.830,160.073
C08120=1015.014,255.486,-136.869,168.804,52.822,160.072
C08121=1015.020,255.735,-136.896,168.809,52.814,160.072
C08122=1015.026,255.983,-136.924,168.813,52.806,160.071
C08123=1015.031,256.232,-136.951,168.818,52.799,160.070
C08124=1015.037,256.480,-136.979,168.823,52.791,160.070
C08125=1015.043,256.729,-137.006,168.828,52.783,160.069
C08126=1015.048,256.977,-137.034,168.833,52.775,160.068
C08127=1015.055,257.225,-137.062,168.838,52.768,160.067
C08128=1015.060,257.474,-137.089,168.843,52.760,160.067
C08129=1015.066,257.722,-137.116,168.849,52.752,160.066
C08130=1015.071,257.971,-137.144,168.854,52.744,160.065
C08131=1015.077,258.219,-137.172,168.859,52.736,160.065
C08132=1015.083,258.467,-137.199,168.864,52.729,160.064
C08133=1015.088,258.716,-137.227,168.869,52.721,160.063
C08134=1015.094,258.964,-137.254,168.874,52.714,160.063
C08135=1015.100,259.212,-137.282,168.879,52.706,160.062
C08136=1015.106,259.460,-137.310,168.884,52.698,160.061
C08137=1015.112,259.709,-137.338,168.889,52.690,160.060
C08138=1015.117,259.957,-137.366,168.895,52.683,160.060
C08139=1015.123,260.205,-137.394,168.900,52.676,160.059
C08140=1015.128,260.453,-137.422,168.905,52.668,160.059
C08141=1015.134,260.702,-137.451,168.910,52.661,160.058
C08142=1015.139,260.951,-137.479,168.915,52.653,160.057
C08143=1015.144,261.199,-137.507,168.920,52.646,160.057
C08144=1015.150,261.447,-137.535,168.925,52.638,160.056
C08145=1015.156,261.695,-137.563,168.930,52.631,160.055
C08146=1015.162,261.944,-137.592,168.935,52.624,160.055
C08147=1015.167,262.192,-137.620,168.940,52.617,160.054
C08148=1015.173,262.441,-137.648,168.945,52.609,160.053
C08149=1015.178,262.689,-137.676,168.951,52.602,160.053
C08150=1015.184,262.929,-137.703,168.956,52.594,160.052
C08151=1015.190,263.168,-137.730,168.960,52.587,160.052
C08152=1015.195,263.408,-137.757,168.965,52.580,160.051
C08153=1015.200,263.647,-137.784,168.971,52.573,160.051
C08154=1015.206,263.887,-137.812,168.975,52.566,160.050
C08155=1015.211,264.127,-137.839,168.980,52.559,160.049
C08156=1015.217,264.366,-137.867,168.986,52.552,160.049
C08157=1015.223,264.606,-137.894,168.990,52.545,160.048
C08158=1015.227,264.854,-137.922,168.996,52.538,160.048
C08159=1015.233,265.103,-137.951,169.001,52.530,160.047
C08160=1015.239,265.350,-137.979,169.006,52.523,160.046
C08161=1015.245,265.599,-138.008,169.011,52.516,160.046
C08162=1015.250,265.847,-138.036,169.016,52.509,160.045
C08163=1015.257,266.095,-138.065,169.021,52.502,160.045
C08164=1015.261,266.344,-138.093,169.026,52.495,160.044
C08165=1015.267,266.592,-138.122,169.032,52.488,160.044
C08166=1015.273,266.840,-138.151,169.037,52.480,160.043
C08167=1015.279,267.089,-138.179,169.042,52.473,160.042
C08168=1015.285,267.337,-138.208,169.048,52.466,160.042
C08169=1015.290,267.585,-138.236,169.052,52.460,160.041
C08170=1015.295,267.834,-138.265,169.057,52.452,160.041
C08171=1015.302,268.082,-138.294,169.063,52.445,160.040
C08172=1015.307,268.330,-138.322,169.068,52.438,160.040
C08173=1015.313,268.578,-138.351,169.073,52.431,160.039
C08174=1015.319,268.827,-138.380,169.079,52.424,160.039
C08175=1015.324,269.075,-138.408,169.083,52.417,160.038
C08176=1015.330,269.323,-138.437,169.089,52.410,160.037
C08177=1015.336,269.572,-138.466,169.094,52.403,160.037
C08178=1015.341,269.819,-138.495,169.099,52.396,160.036
C08179=1015.346,270.068,-138.524,169.105,52.389,160.036
C08180=1015.353,270.316,-138.553,169.109,52.382,160.035
C08181=1015.358,270.564,-138.582,169.115,52.375,160.035
C08182=1015.364,270.813,-138.610,169.120,52.368,160.034
C08183=1015.370,271.061,-138.639,169.126,52.361,160.034
C08184=1015.375,271.308,-138.668,169.131,52.354,160.033
C08185=1015.381,271.558,-138.697,169.136,52.348,160.033
C08186=1015.387,271.806,-138.726,169.142,52.341,160.032
C08187=1015.392,272.054,-138.756,169.147,52.334,160.032
C08188=1015.398,272.302,-138.784,169.152,52.327,160.031
C08189=1015.404,272.550,-138.813,169.157,52.321,160.031
C08190=1015.410,272.799,-138.842,169.162,52.314,160.030
C08191=1015.416,273.047,-138.871,169.168,52.307,160.030
C08192=1015.421,273.295,-138.901,169.174,52.300,160.029
C08193=1015.427,273.543,-138.930,169.178,52.294,160.029
C08194=1015.432,273.791,-138.959,169.184,52.287,160.028
C08195=1015.439,274.039,-138.988,169.189,52.280,160.028
C08196=1015.444,274.288,-139.018,169.195,52.273,160.028
C08197=1015.450,274.536,-139.046,169.199,52.267,160.027
C08198=1015.455,274.784,-139.076,169.205,52.260,160.026
C08199=1015.461,275.032,-139.105,169.211,52.253,160.026
C08200=1015.467,275.281,-139.134,169.215,52.247,160.026
C08201=1015.473,275.529,-139.163,169.221,52.240,160.025
C08202=1015.479,275.777,-139.193,169.227,52.233,160.025
C08203=1015.485,276.026,-139.222,169.232,52.226,160.024
C08204=1015.490,276.274,-139.252,169.237,52.221,160.024
C08205=1015.496,276.521,-139.281,169.242,52.214,160.023
C08206=1015.502,276.769,-139.311,169.248,52.207,160.023
C08207=1015.507,277.018,-139.340,169.253,52.201,160.022
C08208=1015.514,277.266,-139.369,169.259,52.194,160.022
C08209=1015.519,277.514,-139.399,169.264,52.187,160.022
C08210=1015.524,277.756,-139.428,169.269,52.181,160.021
C08211=1015.530,277.997,-139.457,169.275,52.175,160.021
C08212=1015.536,278.239,-139.486,169.279,52.168,160.020
C08213=1015.541,278.481,-139.515,169.284,52.163,160.020
C08214=1015.547,278.723,-139.543,169.290,52.156,160.020
C08215=1015.553,278.965,-139.572,169.295,52.150,160.019
C08216=1015.558,279.206,-139.601,169.301,52.144,160.019
C08217=1015.565,279.449,-139.631,169.305,52.137,160.018
C08218=1015.570,279.697,-139.660,169.311,52.131,160.018
C08219=1015.576,279.945,-139.690,169.317,52.125,160.018
C08220=1015.582,280.193,-139.720,169.322,52.118,160.017
C08221=1015.588,280.441,-139.749,169.328,52.112,160.017
C08222=1015.593,280.690,-139.779,169.334,52.106,160.017
C08223=1015.599,280.938,-139.809,169.338,52.100,160.016
C08224=1015.605,281.186,-139.838,169.344,52.093,160.016
C08225=1015.611,281.434,-139.869,169.350,52.086,160.015
C08226=1015.617,281.682,-139.898,169.355,52.080,160.015
C08227=1015.622,281.931,-139.928,169.361,52.074,160.015
C08228=1015.629,282.178,-139.958,169.365,52.068,160.014
C08229=1015.634,282.426,-139.987,169.371,52.061,160.014
C08230=1015.640,282.674,-140.018,169.377,52.055,160.013
C08231=1015.646,282.922,-140.047,169.382,52.049,160.013
C08232=1015.652,283.170,-140.077,169.388,52.043,160.013
C08233=1015.658,283.419,-140.107,169.394,52.037,160.012
C08234=1015.664,283.667,-140.138,169.399,52.031,160.012
C08235=1015.670,283.915,-140.167,169.405,52.024,160.012
C08236=1015.676,284.163,-140.197,169.410,52.017,160.011
C08237=1015.682,284.411,-140.227,169.415,52.011,160.011
C08238=1015.688,284.659,-140.258,169.421,52.005,160.011
C08239=1015.693,284.907,-140.287,169.426,51.999,160.010
C08240=1015.699,285.155,-140.318,169.432,51.994,160.010
C08241=1015.705,285.404,-140.348,169.438,51.987,160.010
C08242=1015.711,285.651,-140.379,169.443,51.982,160.009
C08243=1015.717,285.900,-140.408,169.449,51.975,160.009
C08244=1015.723,286.148,-140.439,169.454,51.969,160.009
C08245=1015.728,286.395,-140.469,169.460,51.963,160.008
C08246=1015.736,286.644,-140.499,169.465,51.957,160.008
C08247=1015.741,286.892,-140.529,169.471,51.951,160.008
C08248=1015.747,287.139,-140.560,169.476,51.945,160.007
C08249=1015.753,287.387,-140.590,169.482,51.939,160.007
C08250=1015.759,287.635,-140.621,169.488,51.933,160.007
C08251=1015.764,287.884,-140.652,169.493,51.927,160.006
C08252=1015.770,288.132,-140.681,169.499,51.921,160.006
C08253=1015.776,288.380,-140.712,169.504,51.916,160.006
C08254=1015.782,288.629,-140.743,169.510,51.909,160.006
C08255=1015.788,288.876,-140.773,169.516,51.903,160.005
C08256=1015.794,289.124,-140.803,169.521,51.898,160.005
C08257=1015.800,289.373,-140.834,169.527,51.892,160.005
C08258=1015.806,289.620,-140.865,169.532,51.886,160.005
C08259=1015.812,289.868,-140.895,169.538,51.880,160.004
C08260=1015.818,290.116,-140.926,169.543,51.874,160.004
C08261=1015.824,290.364,-140.956,169.549,51.868,160.004
C08262=1015.830,290.612,-140.987,169.555,51.863,160.004
C08263=1015.837,290.860,-141.018,169.560,51.857,160.003
C08264=1015.842,291.108,-141.048,169.567,51.851,160.003
C08265=1015.849,291.356,-141.079,169.572,51.845,160.003
C08266=1015.854,291.604,-141.110,169.578,51.840,160.003
C08267=1015.860,291.852,-141.141,169.583,51.834,160.002
C08268=1015.866,292.100,-141.171,169.589,51.828,160.002
C08269=1015.873,292.348,-141.202,169.594,51.822,160.002
C08270=1015.878,292.596,-141.233,169.601,51.817,160.002
C08271=1015.884,292.844,-141.264,169.606,51.811,160.001
C08272=1015.890,293.092,-141.295,169.612,51.805,160.001
C08273=1015.895,293.340,-141.326,169.617,51.800,160.001
C08274=1015.902,293.588,-141.357,169.624,51.794,160.001
C08275=1015.907,293.836,-141.388,169.629,51.789,160.001
C08276=1015.913,294.083,-141.420,169.635,51.783,160.000
C08277=1015.919,294.331,-141.452,169.640,51.778,160.000
C08278=1015.925,294.579,-141.482,169.646,51.773,160.000
C08279=1015.931,294.827,-141.514,169.652,51.766,160.000
C08280=1015.937,295.075,-141.544,169.657,51.761,160.000
C08281=1015.943,295.323,-141.576,169.663,51.756,160.000
C08282=1015.949,295.571,-141.607,169.669,51.750,159.999
C08283=1015.955,295.819,-141.639,169.675,51.745,159.999
C08284=1015.961,296.067,-141.670,169.680,51.740,159.999
C08285=1015.967,296.315,-141.702,169.687,51.734,159.999
C08286=1015.973,296.563,-141.732,169.692,51.728,159.999
C08287=1015.979,296.811,-141.764,169.698,51.723,159.998
C08288=1015.984,297.058,-141.796,169.703,51.717,159.998
C08289=1015.991,297.306,-141.827,169.709,51.712,159.998
C08290=1015.996,297.555,-141.859,169.715,51.707,159.998
C08291=1016.003,297.802,-141.890,169.720,51.701,159.998
C08292=1016.008,298.051,-141.922,169.727,51.696,159.998
C08293=1016.015,298.298,-141.953,169.732,51.691,159.998
C08294=1016.021,298.546,-141.985,169.739,51.685,159.997
C08295=1016.026,298.794,-142.015,169.744,51.680,159.997
C08296=1016.032,299.042,-142.047,169.750,51.674,159.997
C08297=1016.039,299.290,-142.079,169.756,51.669,159.997
C08298=1016.045,299.537,-142.110,169.762,51.664,159.997
C08299=1016.051,299.785,-142.142,169.767,51.658,159.997
C08300=1016.057,300.034,-142.174,169.774,51.653,159.997
C08301=1016.063,300.281,-142.205,169.780,51.648,159.997
C08302=1016.069,300.529,-142.237,169.785,51.643,159.996
C08303=1016.075,300.777,-142.269,169.791,51.638,159.996
C08304=1016.082,301.025,-142.300,169.797,51.632,159.996
C08305=1016.087,301.273,-142.332,169.803,51.627,159.996
C08306=1016.094,301.520,-142.363,169.809,51.622,159.996
C08307=1016.100,301.769,-142.395,169.815,51.617,159.996
C08308=1016.107,302.017,-142.427,169.821,51.612,159.996
C08309=1016.112,302.264,-142.458,169.827,51.606,159.996
C08310=1016.119,302.512,-142.490,169.832,51.601,159.995
C08311=1016.125,302.760,-142.522,169.839,51.596,159.996
C08312=1016.132,303.008,-142.553,169.844,51.591,159.995
C08313=1016.137,303.256,-142.585,169.851,51.585,159.995
C08314=1016.143,303.503,-142.618,169.857,51.581,159.995
C08315=1016.150,303.751,-142.649,169.863,51.575,159.995
C08316=1016.156,303.999,-142.681,169.868,51.570,159.995
C08317=1016.163,304.247,-142.713,169.875,51.565,159.995
C08318=1016.169,304.495,-142.745,169.880,51.560,159.995
C08319=1016.176,304.743,-142.777,169.887,51.554,159.995
C08320=1016.181,304.990,-142.808,169.893,51.550,159.995
C08321=1016.188,305.238,-142.840,169.899,51.544,159.995
C08322=1016.194,305.486,-142.872,169.905,51.540,159.995
C08323=1016.201,305.734,-142.904,169.911,51.534,159.995
C08324=1016.207,305.982,-142.936,169.916,51.529,159.994
C08325=1016.213,306.230,-142.968,169.923,51.524,159.995
C08326=1016.220,306.477,-143.000,169.929,51.519,159.994
C08327=1016.226,306.726,-143.032,169.935,51.514,159.995
C08328=1016.233,306.973,-143.064,169.941,51.509,159.994
C08329=1016.239,307.221,-143.096,169.948,51.504,159.994
C08330=1016.246,307.487,-143.131,169.954,51.499,159.994
C08331=1016.253,307.753,-143.165,169.960,51.493,159.994
C08332=1016.260,308.019,-143.200,169.967,51.488,159.994
C08333=1016.267,308.284,-143.234,169.974,51.483,159.994
C08334=1016.274,308.532,-143.266,169.979,51.478,159.994
C08335=1016.280,308.780,-143.298,169.986,51.473,159.994
C08336=1016.287,309.028,-143.330,169.991,51.468,159.994
C08337=1016.293,309.275,-143.363,169.998,51.463,159.994
C08338=1016.299,309.523,-143.395,170.004,51.458,159.994
C08339=1016.305,309.771,-143.427,170.010,51.453,159.994
C08340=1016.312,310.019,-143.460,170.016,51.449,159.994
C08341=1016.318,310.266,-143.493,170.022,51.444,159.994
C08342=1016.324,310.514,-143.526,170.029,51.439,159.994
C08343=1016.330,310.762,-143.559,170.035,51.435,159.994
C08344=1016.336,311.009,-143.592,170.041,51.430,159.994
C08345=1016.342,311.257,-143.624,170.047,51.426,159.994
C08346=1016.349,311.505,-143.657,170.053,51.421,159.994
C08347=1016.355,311.752,-143.690,170.060,51.416,159.995
C08348=1016.360,312.000,-143.723,170.066,51.412,159.995
C08349=1016.367,312.248,-143.756,170.071,51.407,159.995
C08350=1016.373,312.495,-143.789,170.078,51.402,159.995
C08351=1016.379,312.743,-143.821,170.084,51.398,159.995
C08352=1016.386,312.991,-143.855,170.091,51.393,159.995
C08353=1016.392,313.239,-143.888,170.096,51.388,159.995
C08354=1016.398,313.486,-143.921,170.103,51.385,159.995
C08355=1016.405,313.734,-143.954,170.110,51.380,159.995
C08356=1016.411,313.981,-143.987,170.115,51.375,159.995
C08357=1016.418,314.229,-144.020,170.122,51.370,159.995
C08358=1016.423,314.477,-144.053,170.128,51.366,159.995
C08359=1016.430,314.725,-144.086,170.135,51.361,159.995
C08360=1016.436,314.972,-144.119,170.141,51.357,159.996
C08361=1016.443,315.220,-144.152,170.147,51.353,159.996
C08362=1016.449,315.468,-144.185,170.153,51.348,159.996
C08363=1016.455,315.716,-144.219,170.159,51.343,159.996
C08364=1016.462,315.963,-144.252,170.166,51.339,159.996
C08365=1016.468,316.211,-144.285,170.172,51.335,159.996
C08366=1016.475,316.459,-144.318,170.178,51.330,159.996
C08367=1016.481,316.706,-144.351,170.185,51.326,159.996
C08368=1016.488,316.954,-144.385,170.191,51.322,159.996
C08369=1016.494,317.202,-144.418,170.198,51.317,159.997
C08370=1016.500,317.449,-144.451,170.204,51.313,159.997
C08371=1016.507,317.697,-144.484,170.211,51.308,159.997
C08372=1016.513,317.944,-144.519,170.217,51.304,159.997
C08373=1016.519,318.192,-144.551,170.224,51.299,159.997
C08374=1016.527,318.440,-144.585,170.230,51.295,159.997
C08375=1016.533,318.687,-144.618,170.236,51.291,159.997
C08376=1016.540,318.935,-144.652,170.243,51.286,159.998
C08377=1016.546,319.183,-144.685,170.249,51.282,159.998
C08378=1016.553,319.430,-144.719,170.256,51.278,159.998
C08379=1016.559,319.678,-144.752,170.262,51.274,159.998
C08380=1016.566,319.926,-144.785,170.269,51.269,159.998
C08381=1016.572,320.174,-144.819,170.275,51.265,159.998
C08382=1016.579,320.421,-144.853,170.282,51.260,159.999
C08383=1016.586,320.668,-144.886,170.288,51.256,159.999
C08384=1016.593,320.917,-144.919,170.295,51.252,159.999
C08385=1016.599,321.163,-144.953,170.301,51.248,159.999
C08386=1016.606,321.411,-144.987,170.308,51.244,159.999
C08387=1016.612,321.659,-145.020,170.314,51.239,159.999
C08388=1016.619,321.907,-145.054,170.321,51.235,160.000
C08389=1016.626,322.154,-145.087,170.327,51.231,160.000
C08390=1016.634,322.426,-145.124,170.334,51.226,160.000
C08391=1016.640,322.696,-145.161,170.341,51.222,160.000
C08392=1016.648,322.969,-145.198,170.349,51.217,160.000
C08393=1016.656,323.239,-145.235,170.356,51.213,160.001
C08394=1016.662,323.487,-145.268,170.362,51.209,160.001
C08395=1016.669,323.735,-145.302,170.369,51.204,160.001
C08396=1016.676,323.982,-145.336,170.375,51.200,160.001
C08397=1016.682,324.230,-145.370,170.383,51.196,160.002
C08398=1016.689,324.477,-145.404,170.389,51.192,160.002
C08399=1016.697,324.725,-145.437,170.396,51.188,160.002
C08400=1016.703,324.972,-145.471,170.402,51.184,160.002
C08401=1016.710,325.220,-145.505,170.409,51.179,160.002
C08402=1016.717,325.468,-145.539,170.415,51.176,160.003
C08403=1016.724,325.715,-145.573,170.422,51.171,160.003
C08404=1016.731,325.962,-145.606,170.430,51.167,160.003
C08405=1016.737,326.210,-145.641,170.436,51.164,160.004
C08406=1016.744,326.458,-145.675,170.442,51.160,160.004
C08407=1016.751,326.705,-145.710,170.449,51.156,160.004
C08408=1016.757,326.953,-145.744,170.456,51.152,160.004
C08409=1016.764,327.200,-145.778,170.463,51.148,160.005
C08410=1016.771,327.448,-145.813,170.469,51.144,160.005
C08411=1016.777,327.696,-145.847,170.477,51.140,160.005
C08412=1016.785,327.943,-145.881,170.483,51.136,160.005
C08413=1016.791,328.191,-145.916,170.490,51.132,160.006
C08414=1016.797,328.438,-145.950,170.496,51.128,160.006
C08415=1016.804,328.686,-145.985,170.504,51.125,160.007
C08416=1016.811,328.933,-146.019,170.510,51.121,160.007
C08417=1016.818,329.181,-146.054,170.517,51.117,160.007
C08418=1016.824,329.428,-146.089,170.524,51.114,160.007
C08419=1016.832,329.676,-146.123,170.531,51.110,160.008
C08420=1016.838,329.923,-146.158,170.537,51.106,160.008
C08421=1016.845,330.171,-146.192,170.545,51.102,160.009
C08422=1016.852,330.418,-146.227,170.551,51.098,160.009
C08423=1016.859,330.666,-146.262,170.558,51.094,160.009
C08424=1016.866,330.914,-146.296,170.565,51.091,160.009
C08425=1016.873,331.161,-146.331,170.572,51.087,160.010
C08426=1016.880,331.409,-146.365,170.579,51.084,160.010
C08427=1016.886,331.656,-146.400,170.586,51.080,160.010
C08428=1016.894,331.903,-146.435,170.592,51.076,160.011
C08429=1016.900,332.151,-146.469,170.600,51.072,160.011
C08430=1016.907,332.399,-146.504,170.606,51.069,160.011
C08431=1016.914,332.646,-146.540,170.614,51.065,160.012
C08432=1016.921,332.893,-146.575,170.620,51.062,160.012
C08433=1016.927,333.141,-146.610,170.627,51.058,160.013
C08434=1016.934,333.388,-146.645,170.634,51.055,160.013
C08435=1016.941,333.635,-146.680,170.642,51.051,160.014
C08436=1016.948,333.882,-146.715,170.648,51.047,160.014
C08437=1016.955,334.130,-146.750,170.655,51.044,160.014
C08438=1016.962,334.377,-146.785,170.662,51.041,160.015
C08439=1016.969,334.625,-146.820,170.669,51.036,160.015
C08440=1016.976,334.873,-146.856,170.676,51.033,160.015
C08441=1016.983,335.120,-146.891,170.683,51.030,160.016
C08442=1016.990,335.367,-146.926,170.690,51.027,160.016
C08443=1016.996,335.615,-146.961,170.697,51.022,160.017
C08444=1017.003,335.862,-146.996,170.704,51.019,160.017
C08445=1017.010,336.110,-147.032,170.711,51.016,160.018
C08446=1017.017,336.357,-147.067,170.718,51.013,160.018
C08447=1017.024,336.605,-147.102,170.726,51.009,160.019
C08448=1017.031,336.852,-147.138,170.732,51.006,160.019
C08449=1017.038,337.100,-147.173,170.740,51.002,160.019
C08450=1017.046,337.366,-147.211,170.747,50.998,160.020
C08451=1017.053,337.634,-147.249,170.755,50.995,160.020
C08452=1017.061,337.900,-147.287,170.762,50.991,160.021
C08453=1017.069,338.167,-147.326,170.771,50.987,160.021
C08454=1017.076,338.414,-147.361,170.778,50.984,160.022
C08455=1017.083,338.662,-147.396,170.785,50.981,160.022
C08456=1017.090,338.909,-147.432,170.792,50.978,160.023
C08457=1017.096,339.157,-147.468,170.799,50.974,160.023
C08458=1017.104,339.404,-147.504,170.806,50.971,160.024
C08459=1017.111,339.652,-147.539,170.814,50.968,160.024
C08460=1017.118,339.898,-147.575,170.821,50.965,160.025
C08461=1017.125,340.146,-147.611,170.828,50.961,160.025
C08462=1017.132,340.393,-147.647,170.836,50.958,160.026
C08463=1017.139,340.641,-147.683,170.842,50.955,160.026
C08464=1017.146,340.888,-147.719,170.850,50.952,160.027
C08465=1017.153,341.135,-147.754,170.857,50.949,160.027
C08466=1017.161,341.382,-147.791,170.865,50.945,160.028
C08467=1017.167,341.630,-147.826,170.872,50.943,160.028
C08468=1017.175,341.878,-147.863,170.879,50.939,160.029
C08469=1017.182,342.124,-147.898,170.887,50.936,160.029
C08470=1017.189,342.372,-147.935,170.894,50.933,160.030
C08471=1017.196,342.619,-147.970,170.902,50.930,160.031
C08472=1017.203,342.867,-148.007,170.908,50.926,160.031
C08473=1017.210,343.114,-148.042,170.916,50.924,160.032
C08474=1017.218,343.361,-148.079,170.924,50.920,160.032
C08475=1017.225,343.609,-148.115,170.931,50.918,160.033
C08476=1017.232,343.856,-148.151,170.938,50.914,160.033
C08477=1017.239,344.103,-148.188,170.945,50.912,160.034
C08478=1017.246,344.350,-148.224,170.953,50.908,160.034
C08479=1017.254,344.597,-148.260,170.961,50.905,160.035
C08480=1017.261,344.845,-148.296,170.968,50.903,160.036
C08481=1017.268,345.092,-148.332,170.976,50.899,160.036
C08482=1017.275,345.339,-148.369,170.984,50.896,160.037
C08483=1017.283,345.587,-148.405,170.990,50.893,160.037
C08484=1017.290,345.834,-148.441,170.998,50.890,160.038
C08485=1017.297,346.081,-148.478,171.005,50.888,160.039
C08486=1017.305,346.328,-148.515,171.013,50.884,160.039
C08487=1017.313,346.576,-148.551,171.021,50.881,160.040
C08488=1017.319,346.823,-148.588,171.028,50.879,160.041
C08489=1017.327,347.070,-148.624,171.036,50.876,160.041
C08490=1017.334,347.317,-148.661,171.043,50.873,160.042
C08491=1017.341,347.565,-148.697,171.050,50.870,160.042
C08492=1017.348,347.812,-148.734,171.058,50.867,160.043
C08493=1017.356,348.059,-148.771,171.066,50.864,160.044
C08494=1017.363,348.306,-148.808,171.073,50.862,160.045
C08495=1017.371,348.553,-148.845,171.081,50.859,160.045
C08496=1017.378,348.801,-148.881,171.090,50.856,160.046
C08497=1017.385,349.047,-148.918,171.097,50.854,160.047
C08498=1017.392,349.295,-148.955,171.105,50.851,160.047
C08499=1017.400,349.542,-148.992,171.113,50.848,160.048
C08500=1017.407,349.789,-149.029,171.120,50.845,160.049
C08501=1017.415,350.036,-149.065,171.128,50.842,160.049
C08502=1017.422,350.283,-149.103,171.136,50.840,160.050
C08503=1017.429,350.531,-149.140,171.144,50.837,160.051
C08504=1017.437,350.778,-149.177,171.151,50.834,160.051
C08505=1017.444,351.025,-149.214,171.159,50.831,160.052
C08506=1017.452,351.272,-149.251,171.167,50.829,160.053
C08507=1017.459,351.520,-149.288,171.174,50.827,160.054
C08508=1017.467,351.766,-149.325,171.182,50.824,160.054
C08509=1017.474,352.014,-149.362,171.190,50.821,160.055
C08510=1017.482,352.278,-149.402,171.198,50.818,160.056
C08511=1017.490,352.541,-149.441,171.206,50.816,160.057
C08512=1017.499,352.806,-149.481,171.215,50.813,160.057
C08513=1017.506,353.070,-149.521,171.223,50.810,160.058
C08514=1017.514,353.318,-149.558,171.231,50.807,160.059
C08515=1017.521,353.565,-149.596,171.240,50.805,160.060
C08516=1017.529,353.812,-149.633,171.247,50.802,160.060
C08517=1017.537,354.059,-149.670,171.255,50.800,160.061
C08518=1017.544,354.305,-149.709,171.263,50.797,160.062
C08519=1017.551,354.553,-149.746,171.272,50.795,160.063
C08520=1017.559,354.799,-149.783,171.279,50.792,160.064
C08521=1017.567,355.047,-149.821,171.287,50.790,160.064
C08522=1017.575,355.294,-149.859,171.295,50.787,160.065
C08523=1017.582,355.542,-149.896,171.303,50.785,160.066
C08524=1017.590,355.788,-149.934,171.311,50.782,160.067
C08525=1017.597,356.035,-149.971,171.319,50.780,160.068
C08526=1017.605,356.282,-150.009,171.327,50.777,160.068
C08527=1017.613,356.529,-150.047,171.335,50.775,160.069
C08528=1017.621,356.776,-150.084,171.344,50.773,160.070
C08529=1017.628,357.023,-150.122,171.352,50.770,160.071
C08530=1017.635,357.270,-150.160,171.360,50.768,160.072
C08531=1017.643,357.518,-150.198,171.367,50.766,160.073
C08532=1017.651,357.764,-150.236,171.376,50.764,160.074
C08533=1017.658,358.011,-150.274,171.384,50.761,160.074
C08534=1017.667,358.258,-150.312,171.392,50.759,160.075
C08535=1017.674,358.505,-150.349,171.401,50.756,160.076
C08536=1017.682,358.752,-150.388,171.409,50.754,160.077
C08537=1017.690,359.000,-150.425,171.417,50.752,160.078
C08538=1017.697,359.246,-150.464,171.425,50.750,160.079
C08539=1017.705,359.493,-150.502,171.433,50.748,160.080
C08540=1017.713,359.740,-150.541,171.442,50.746,160.081
C08541=1017.720,359.987,-150.578,171.450,50.743,160.081
C08542=1017.728,360.234,-150.617,171.458,50.741,160.082
C08543=1017.736,360.481,-150.655,171.467,50.739,160.083
C08544=1017.744,360.728,-150.693,171.475,50.737,160.084
C08545=1017.752,360.974,-150.732,171.484,50.734,160.085
C08546=1017.760,361.222,-150.770,171.491,50.732,160.086
C08547=1017.767,361.468,-150.809,171.499,50.730,160.087
C08548=1017.775,361.716,-150.848,171.508,50.728,160.088
C08549=1017.782,361.962,-150.886,171.517,50.726,160.089
C08550=1017.790,362.209,-150.925,171.525,50.724,160.090
C08551=1017.798,362.456,-150.963,171.533,50.722,160.091
C08552=1017.806,362.703,-151.001,171.542,50.720,160.092
C08553=1017.814,362.950,-151.040,171.551,50.718,160.093
C08554=1017.822,363.197,-151.078,171.559,50.716,160.094
C08555=1017.830,363.443,-151.118,171.567,50.714,160.095
C08556=1017.838,363.690,-151.156,171.576,50.711,160.095
C08557=1017.846,363.937,-151.195,171.585,50.710,160.097
C08558=1017.854,364.184,-151.233,171.593,50.707,160.098
C08559=1017.861,364.431,-151.273,171.602,50.706,160.099
C08560=1017.869,364.678,-151.311,171.610,50.704,160.100
C08561=1017.877,364.925,-151.350,171.619,50.702,160.101
C08562=1017.886,365.172,-151.389,171.627,50.700,160.102
C08563=1017.893,365.418,-151.427,171.636,50.698,160.102
C08564=1017.902,365.665,-151.466,171.645,50.696,160.104
C08565=1017.910,365.912,-151.505,171.653,50.694,160.105
C08566=1017.918,366.159,-151.544,171.662,50.692,160.106
C08567=1017.926,366.405,-151.583,171.670,50.690,160.107
C08568=1017.934,366.652,-151.622,171.679,50.688,160.108
C08569=1017.942,366.899,-151.661,171.688,50.687,160.109
C08570=1017.952,367.171,-151.704,171.697,50.685,160.110
C08571=1017.960,367.442,-151.747,171.707,50.683,160.111
C08572=1017.969,367.715,-151.790,171.717,50.681,160.112
C08573=1017.978,367.986,-151.833,171.727,50.679,160.114
C08574=1017.986,368.233,-151.873,171.735,50.676,160.115
C08575=1017.994,368.480,-151.913,171.744,50.675,160.116
C08576=1018.002,368.726,-151.952,171.753,50.673,160.117
C08577=1018.010,368.973,-151.992,171.762,50.672,160.118
C08578=1018.019,369.220,-152.031,171.770,50.670,160.119
C08579=1018.026,369.467,-152.071,171.779,50.668,160.120
C08580=1018.035,369.713,-152.110,171.788,50.667,160.121
C08581=1018.043,369.960,-152.150,171.798,50.665,160.122
C08582=1018.051,370.207,-152.190,171.807,50.663,160.124
C08583=1018.059,370.453,-152.229,171.815,50.661,160.125
C08584=1018.067,370.700,-152.269,171.824,50.660,160.126
C08585=1018.076,370.947,-152.308,171.833,50.658,160.127
C08586=1018.083,371.194,-152.348,171.842,50.657,160.128
C08587=1018.092,371.440,-152.388,171.851,50.656,160.129
C08588=1018.100,371.686,-152.428,171.861,50.654,160.131
C08589=1018.108,371.933,-152.467,171.869,50.652,160.132
C08590=1018.117,372.180,-152.507,171.878,50.650,160.133
C08591=1018.125,372.427,-152.547,171.887,50.649,160.134
C08592=1018.134,372.673,-152.587,171.896,50.648,160.135
C08593=1018.141,372.920,-152.627,171.906,50.646,160.137
C08594=1018.150,373.167,-152.666,171.915,50.644,160.138
C08595=1018.159,373.413,-152.707,171.924,50.643,160.139
C08596=1018.167,373.660,-152.747,171.933,50.641,160.140
C08597=1018.176,373.906,-152.787,171.943,50.640,160.142
C08598=1018.183,374.153,-152.827,171.952,50.638,160.143
C08599=1018.193,374.400,-152.867,171.960,50.637,160.144
C08600=1018.201,374.647,-152.907,171.971,50.635,160.145
C08601=1018.209,374.893,-152.947,171.979,50.634,160.146
C08602=1018.219,375.139,-152.987,171.989,50.633,160.148
C08603=1018.226,375.386,-153.027,171.998,50.631,160.149
C08604=1018.235,375.632,-153.067,172.008,50.630,160.150
C08605=1018.244,375.879,-153.108,172.017,50.629,160.151
C08606=1018.252,376.126,-153.148,172.027,50.627,160.153
C08607=1018.261,376.373,-153.189,172.036,50.626,160.154
C08608=1018.269,376.619,-153.229,172.045,50.625,160.155
C08609=1018.277,376.865,-153.270,172.055,50.623,160.157
C08610=1018.286,377.112,-153.311,172.064,50.622,160.158
C08611=1018.294,377.358,-153.351,172.073,50.621,160.159
C08612=1018.303,377.605,-153.392,172.083,50.619,160.161
C08613=1018.311,377.852,-153.433,172.092,50.618,160.162
C08614=1018.320,378.098,-153.474,172.102,50.617,160.163
C08615=1018.328,378.344,-153.515,172.112,50.616,160.165
C08616=1018.337,378.591,-153.555,172.121,50.615,160.166
C08617=1018.345,378.837,-153.596,172.131,50.613,160.167
C08618=1018.354,379.084,-153.637,172.140,50.612,160.169
C08619=1018.362,379.330,-153.678,172.149,50.611,160.170
C08620=1018.372,379.577,-153.719,172.160,50.610,160.172
C08621=1018.380,379.824,-153.760,172.169,50.609,160.173
C08622=1018.389,380.069,-153.801,172.179,50.608,160.174
C08623=1018.397,380.316,-153.842,172.188,50.606,160.176
C08624=1018.407,380.563,-153.883,172.198,50.605,160.177
C08625=1018.415,380.809,-153.924,172.208,50.605,160.179
C08626=1018.424,381.056,-153.965,172.218,50.603,160.180
C08627=1018.432,381.302,-154.007,172.227,50.602,160.181
C08628=1018.441,381.549,-154.048,172.237,50.601,160.183
C08629=1018.450,381.794,-154.088,172.247,50.600,160.184
C08630=1018.460,382.089,-154.138,172.259,50.598,160.186
C08631=1018.471,382.383,-154.187,172.271,50.597,160.188
C08632=1018.482,382.677,-154.237,172.283,50.597,160.189
C08633=1018.492,382.971,-154.286,172.294,50.595,160.191
C08634=1018.502,383.218,-154.326,172.304,50.594,160.193
C08635=1018.510,383.464,-154.368,172.315,50.593,160.194
C08636=1018.519,383.710,-154.410,172.324,50.592,160.196
C08637=1018.528,383.957,-154.452,172.335,50.591,160.197
C08638=1018.538,384.203,-154.493,172.345,50.590,160.199
C08639=1018.547,384.449,-154.534,172.354,50.590,160.200
C08640=1018.556,384.695,-154.576,172.365,50.588,160.202
C08641=1018.564,384.942,-154.617,172.375,50.587,160.203
C08642=1018.573,385.189,-154.659,172.385,50.587,160.205
C08643=1018.583,385.434,-154.701,172.395,50.586,160.206
C08644=1018.592,385.681,-154.743,172.405,50.585,160.208
C08645=1018.601,385.927,-154.785,172.415,50.584,160.209
C08646=1018.609,386.174,-154.826,172.426,50.584,160.211
C08647=1018.619,386.419,-154.869,172.436,50.583,160.213
C08648=1018.628,386.666,-154.911,172.447,50.582,160.214
C08649=1018.637,386.912,-154.952,172.456,50.581,160.216
C08650=1018.646,387.158,-154.995,172.466,50.580,160.217
C08651=1018.655,387.405,-155.037,172.477,50.579,160.219
C08652=1018.664,387.651,-155.078,172.488,50.578,160.220
C08653=1018.674,387.897,-155.121,172.499,50.578,160.222
C08654=1018.682,388.143,-155.163,172.508,50.578,160.224
C08655=1018.692,388.389,-155.205,172.519,50.577,160.225
C08656=1018.702,388.636,-155.248,172.529,50.576,160.227
C08657=1018.710,388.882,-155.290,172.540,50.575,160.229
C08658=1018.719,389.128,-155.333,172.550,50.575,160.230
C08659=1018.728,389.374,-155.375,172.561,50.574,160.232
C08660=1018.738,389.621,-155.417,172.571,50.574,160.234
C08661=1018.747,389.867,-155.460,172.581,50.573,160.235
C08662=1018.756,390.112,-155.502,172.592,50.572,160.237
C08663=1018.765,390.359,-155.545,172.603,50.572,160.239
C08664=1018.775,390.605,-155.588,172.613,50.571,160.240
C08665=1018.784,390.850,-155.630,172.624,50.571,160.242
C08666=1018.794,391.097,-155.673,172.635,50.570,160.244
C08667=1018.803,391.343,-155.715,172.646,50.570,160.246
C08668=1018.813,391.589,-155.758,172.657,50.569,160.247
C08669=1018.821,391.835,-155.801,172.667,50.569,160.249
C08670=1018.831,392.082,-155.844,172.678,50.568,160.251
C08671=1018.840,392.327,-155.887,172.689,50.568,160.253
C08672=1018.850,392.574,-155.929,172.700,50.567,160.254
C08673=1018.859,392.820,-155.972,172.711,50.567,160.256
C08674=1018.869,393.066,-156.016,172.721,50.567,160.258
C08675=1018.877,393.312,-156.059,172.732,50.566,160.260
C08676=1018.887,393.558,-156.102,172.743,50.566,160.261
C08677=1018.897,393.804,-156.145,172.754,50.565,160.263
C08678=1018.906,394.050,-156.188,172.765,50.565,160.265
C08679=1018.916,394.296,-156.232,172.776,50.565,160.267
C08680=1018.926,394.542,-156.275,172.787,50.565,160.269
C08681=1018.935,394.788,-156.318,172.799,50.564,160.271
C08682=1018.945,395.034,-156.362,172.810,50.564,160.272
C08683=1018.955,395.280,-156.405,172.821,50.563,160.274
C08684=1018.963,395.525,-156.448,172.832,50.563,160.276
C08685=1018.973,395.772,-156.491,172.843,50.563,160.278
C08686=1018.983,396.018,-156.535,172.853,50.563,160.280
C08687=1018.993,396.264,-156.579,172.865,50.562,160.282
C08688=1019.003,396.510,-156.622,172.876,50.562,160.284
C08689=1019.012,396.756,-156.666,172.888,50.562,160.286
C08690=1019.025,397.087,-156.725,172.903,50.562,160.288
C08691=1019.039,397.419,-156.784,172.918,50.562,160.291
C08692=1019.051,397.750,-156.843,172.934,50.561,160.293
C08693=1019.065,398.082,-156.902,172.949,50.561,160.296
C08694=1019.075,398.328,-156.945,172.960,50.561,160.298
C08695=1019.085,398.574,-156.990,172.972,50.561,160.300
C08696=1019.094,398.820,-157.034,172.983,50.561,160.302
C08697=1019.104,399.066,-157.078,172.995,50.560,160.304
C08698=1019.114,399.312,-157.122,173.007,50.561,160.306
C08699=1019.124,399.557,-157.166,173.018,50.560,160.308
C08700=1019.134,399.803,-157.210,173.030,50.560,160.310
C08701=1019.143,400.049,-157.255,173.041,50.561,160.312
C08702=1019.153,400.295,-157.298,173.053,50.560,160.314
C08703=1019.163,400.541,-157.342,173.065,50.560,160.316
C08704=1019.173,400.786,-157.387,173.076,50.561,160.318
C08705=1019.184,401.032,-157.432,173.088,50.561,160.320
C08706=1019.193,401.278,-157.476,173.100,50.561,160.322
C08707=1019.203,401.524,-157.521,173.112,50.561,160.324
C08708=1019.212,401.769,-157.566,173.123,50.561,160.326
C08709=1019.223,402.015,-157.610,173.136,50.561,160.328
C08710=1019.233,402.261,-157.655,173.147,50.562,160.331
C08711=1019.243,402.507,-157.699,173.159,50.562,160.333
C08712=1019.252,402.752,-157.744,173.172,50.561,160.335
C08713=1019.263,402.998,-157.789,173.183,50.562,160.337
C08714=1019.273,403.244,-157.833,173.195,50.562,160.339
C08715=1019.283,403.489,-157.878,173.207,50.562,160.341
C08716=1019.293,403.736,-157.923,173.219,50.562,160.343
C08717=1019.304,403.981,-157.968,173.232,50.563,160.346
C08718=1019.314,404.226,-158.014,173.243,50.563,160.348
C08719=1019.324,404.472,-158.058,173.255,50.563,160.350
C08720=1019.334,404.718,-158.104,173.268,50.563,160.352
C08721=1019.345,404.963,-158.148,173.279,50.564,160.354
C08722=1019.355,405.209,-158.194,173.292,50.563,160.356
C08723=1019.365,405.454,-158.239,173.305,50.564,160.359
C08724=1019.375,405.701,-158.284,173.317,50.564,160.361
C08725=1019.386,405.945,-158.329,173.330,50.564,160.363
C08726=1019.396,406.191,-158.374,173.341,50.565,160.365
C08727=1019.407,406.438,-158.419,173.354,50.565,160.367
C08728=1019.417,406.682,-158.465,173.366,50.566,160.370
C08729=1019.428,406.928,-158.510,173.379,50.566,160.372
C08730=1019.438,407.174,-158.555,173.391,50.566,160.374
C08731=1019.449,407.420,-158.601,173.404,50.567,160.377
C08732=1019.459,407.665,-158.646,173.417,50.567,160.379
C08733=1019.470,407.910,-158.691,173.429,50.567,160.381
C08734=1019.481,408.156,-158.737,173.442,50.568,160.384
C08735=1019.491,408.402,-158.783,173.455,50.568,160.386
C08736=1019.502,408.648,-158.828,173.467,50.568,160.388
C08737=1019.512,408.893,-158.874,173.480,50.569,160.391
C08738=1019.523,409.139,-158.920,173.493,50.569,160.393
C08739=1019.534,409.385,-158.966,173.506,50.570,160.395
C08740=1019.544,409.630,-159.012,173.518,50.570,160.398
C08741=1019.555,409.875,-159.058,173.532,50.571,160.400
C08742=1019.566,410.121,-159.104,173.544,50.572,160.403
C08743=1019.576,410.366,-159.150,173.557,50.572,160.405
C08744=1019.587,410.612,-159.196,173.570,50.573,160.407
C08745=1019.598,410.857,-159.243,173.583,50.574,160.410
C08746=1019.608,411.103,-159.289,173.596,50.574,160.412
C08747=1019.618,411.348,-159.335,173.609,50.575,160.415
C08748=1019.629,411.593,-159.382,173.622,50.576,160.417
C08749=1019.641,411.840,-159.428,173.636,50.577,160.420
C08750=1019.651,412.082,-159.474,173.648,50.577,160.422
C08751=1019.662,412.326,-159.520,173.661,50.578,160.425
C08752=1019.672,412.569,-159.566,173.674,50.579,160.427
C08753=1019.684,412.812,-159.613,173.688,50.579,160.430
C08754=1019.695,413.056,-159.658,173.701,50.580,160.432
C08755=1019.706,413.299,-159.704,173.714,50.581,160.435
C08756=1019.716,413.543,-159.751,173.727,50.582,160.437
C08757=1019.728,413.786,-159.798,173.741,50.582,160.440
C08758=1019.738,414.031,-159.844,173.754,50.583,160.442
C08759=1019.749,414.276,-159.890,173.767,50.584,160.445
C08760=1019.761,414.522,-159.937,173.781,50.584,160.447
C08761=1019.772,414.767,-159.984,173.794,50.585,160.450
C08762=1019.783,415.013,-160.031,173.809,50.586,160.453
C08763=1019.793,415.258,-160.078,173.822,50.587,160.455
C08764=1019.805,415.503,-160.126,173.836,50.588,160.458
C08765=1019.816,415.748,-160.172,173.849,50.589,160.460
C08766=1019.827,415.994,-160.220,173.863,50.590,160.463
C08767=1019.839,416.239,-160.268,173.877,50.591,160.466
C08768=1019.849,416.484,-160.315,173.891,50.592,160.469
C08769=1019.861,416.730,-160.362,173.905,50.593,160.471
C08770=1019.872,416.975,-160.410,173.918,50.594,160.474
C08771=1019.883,417.220,-160.457,173.933,50.595,160.477
C08772=1019.894,417.465,-160.504,173.947,50.596,160.480
C08773=1019.906,417.711,-160.552,173.961,50.597,160.482
C08774=1019.917,417.957,-160.600,173.975,50.598,160.485
C08775=1019.928,418.201,-160.647,173.989,50.599,160.488
C08776=1019.940,418.446,-160.695,174.003,50.600,160.491
C08777=1019.951,418.691,-160.743,174.017,50.601,160.493
C08778=1019.963,418.937,-160.790,174.031,50.602,160.496
C08779=1019.975,419.182,-160.838,174.046,50.603,160.499
C08780=1019.986,419.427,-160.886,174.060,50.604,160.502
C08781=1019.998,419.672,-160.934,174.074,50.605,160.505
C08782=1020.009,419.917,-160.981,174.089,50.606,160.508
C08783=1020.020,420.163,-161.030,174.103,50.608,160.510
C08784=1020.032,420.408,-161.077,174.118,50.609,160.513
C08785=1020.044,420.652,-161.126,174.133,50.610,160.516
C08786=1020.056,420.898,-161.174,174.147,50.611,160.519
C08787=1020.067,421.143,-161.222,174.162,50.612,160.522
C08788=1020.078,421.388,-161.270,174.176,50.614,160.525
C08789=1020.091,421.633,-161.319,174.191,50.615,160.528
C08790=1020.102,421.879,-161.367,174.205,50.616,160.531
C08791=1020.114,422.123,-161.416,174.220,50.618,160.534
C08792=1020.126,422.368,-161.465,174.235,50.619,160.537
C08793=1020.138,422.613,-161.512,174.249,50.620,160.540
C08794=1019.763,420.642,-161.462,174.118,50.680,160.534
C08795=1019.751,420.397,-161.414,174.104,50.679,160.531
C08796=1019.740,420.152,-161.366,174.089,50.678,160.528
C08797=1019.728,419.907,-161.318,174.075,50.676,160.525
C08798=1019.717,419.661,-161.270,174.060,50.676,160.522
C08799=1019.705,419.416,-161.222,174.046,50.675,160.520
C08800=1019.693,419.171,-161.174,174.031,50.674,160.517
C08801=1019.682,418.926,-161.126,174.017,50.673,160.514
C08802=1019.670,418.681,-161.078,174.003,50.672,160.511
C08803=1019.658,418.436,-161.031,173.988,50.671,160.508
C08804=1019.648,418.190,-160.984,173.975,50.670,160.506
C08805=1019.636,417.945,-160.936,173.961,50.669,160.503
C08806=1019.624,417.700,-160.888,173.946,50.668,160.500
C08807=1019.614,417.454,-160.841,173.932,50.667,160.497
C08808=1019.602,417.210,-160.793,173.918,50.666,160.495
C08809=1019.591,416.964,-160.746,173.905,50.665,160.492
C08810=1019.580,416.719,-160.698,173.890,50.665,160.489
C08811=1019.568,416.473,-160.651,173.876,50.663,160.486
C08812=1019.557,416.229,-160.604,173.863,50.662,160.484
C08813=1019.546,415.983,-160.556,173.849,50.662,160.481
C08814=1019.535,415.738,-160.509,173.835,50.661,160.478
C08815=1019.523,415.493,-160.462,173.821,50.660,160.476
C08816=1019.513,415.248,-160.414,173.807,50.660,160.473
C08817=1019.502,415.002,-160.367,173.794,50.659,160.471
C08818=1019.491,414.757,-160.321,173.780,50.658,160.468
C08819=1019.479,414.511,-160.274,173.767,50.657,160.465
C08820=1019.468,414.266,-160.227,173.753,50.656,160.463
C08821=1019.457,414.021,-160.180,173.740,50.656,160.460
C08822=1019.447,413.775,-160.133,173.726,50.655,160.458
C08823=1019.436,413.545,-160.089,173.713,50.655,160.455
C08824=1019.426,413.315,-160.046,173.700,50.654,160.453
C08825=1019.416,413.085,-160.002,173.688,50.653,160.450
C08826=1019.405,412.855,-159.958,173.676,50.653,160.448
C08827=1019.395,412.625,-159.915,173.663,50.652,160.446
C08828=1019.385,412.394,-159.872,173.650,50.652,160.443
C08829=1019.375,412.164,-159.828,173.638,50.651,160.441
C08830=1019.364,411.934,-159.784,173.626,50.650,160.439
C08831=1019.353,411.689,-159.738,173.613,50.650,160.436
C08832=1019.343,411.443,-159.692,173.599,50.650,160.434
C08833=1019.332,411.197,-159.646,173.586,50.649,160.431
C08834=1019.321,410.952,-159.599,173.573,50.648,160.429
C08835=1019.310,410.706,-159.553,173.560,50.648,160.427
C08836=1019.299,410.461,-159.507,173.548,50.648,160.424
C08837=1019.288,410.216,-159.461,173.534,50.647,160.422
C08838=1019.278,409.970,-159.414,173.521,50.646,160.419
C08839=1019.268,409.724,-159.368,173.508,50.646,160.417
C08840=1019.257,409.478,-159.322,173.495,50.646,160.415
C08841=1019.247,409.233,-159.276,173.483,50.645,160.412
C08842=1019.237,408.988,-159.231,173.470,50.645,160.410
C08843=1019.226,408.742,-159.185,173.457,50.644,160.407
C08844=1019.215,408.497,-159.139,173.444,50.644,160.405
C08845=1019.204,408.252,-159.094,173.431,50.644,160.403
C08846=1019.194,408.005,-159.049,173.418,50.644,160.401
C08847=1019.183,407.760,-159.003,173.406,50.643,160.398
C08848=1019.172,407.514,-158.957,173.393,50.643,160.396
C08849=1019.162,407.268,-158.912,173.381,50.643,160.394
C08850=1019.151,407.023,-158.867,173.368,50.642,160.391
C08851=1019.141,406.778,-158.821,173.355,50.642,160.389
C08852=1019.130,406.532,-158.776,173.343,50.642,160.387
C08853=1019.121,406.286,-158.731,173.331,50.642,160.385
C08854=1019.109,406.041,-158.685,173.319,50.641,160.382
C08855=1019.099,405.795,-158.640,173.306,50.641,160.380
C08856=1019.089,405.550,-158.595,173.294,50.641,160.378
C08857=1019.079,405.303,-158.549,173.281,50.641,160.376
C08858=1019.068,405.058,-158.505,173.269,50.641,160.374
C08859=1019.058,404.813,-158.459,173.256,50.641,160.371
C08860=1019.047,404.566,-158.414,173.245,50.640,160.369
C08861=1019.038,404.321,-158.369,173.232,50.640,160.367
C08862=1019.027,404.076,-158.325,173.220,50.640,160.365
C08863=1019.017,403.829,-158.280,173.208,50.640,160.363
C08864=1019.007,403.584,-158.235,173.196,50.640,160.361
C08865=1018.997,403.338,-158.190,173.184,50.640,160.358
C08866=1018.986,403.093,-158.146,173.172,50.640,160.356
C08867=1018.977,402.847,-158.101,173.159,50.640,160.354
C08868=1018.966,402.601,-158.056,173.148,50.640,160.352
C08869=1018.957,402.355,-158.011,173.136,50.640,160.350
C08870=1018.946,402.110,-157.967,173.124,50.640,160.348
C08871=1018.936,401.865,-157.922,173.112,50.640,160.346
C08872=1018.926,401.618,-157.877,173.100,50.640,160.344
C08873=1018.917,401.372,-157.832,173.088,50.640,160.342
C08874=1018.906,401.127,-157.788,173.076,50.640,160.339
C08875=1018.897,400.881,-157.744,173.065,50.640,160.338
C08876=1018.887,400.635,-157.699,173.053,50.640,160.335
C08877=1018.878,400.389,-157.655,173.041,50.640,160.333
C08878=1018.867,400.143,-157.611,173.029,50.640,160.331
C08879=1018.857,399.897,-157.566,173.018,50.640,160.329
C08880=1018.847,399.652,-157.522,173.006,50.641,160.327
C08881=1018.837,399.406,-157.478,172.995,50.640,160.325
C08882=1018.827,399.160,-157.435,172.983,50.641,160.323
C08883=1018.817,398.915,-157.390,172.971,50.641,160.321
C08884=1018.808,398.668,-157.346,172.959,50.641,160.319
C08885=1018.798,398.423,-157.302,172.948,50.642,160.318
C08886=1018.788,398.176,-157.258,172.936,50.642,160.315
C08887=1018.776,397.843,-157.199,172.921,50.642,160.313
C08888=1018.762,397.508,-157.139,172.906,50.642,160.310
C08889=1018.749,397.175,-157.080,172.890,50.643,160.308
C08890=1018.736,396.841,-157.021,172.875,50.643,160.305
C08891=1018.726,396.595,-156.977,172.863,50.644,160.303
C08892=1018.716,396.349,-156.934,172.852,50.644,160.301
C08893=1018.706,396.103,-156.890,172.841,50.644,160.300
C08894=1018.696,395.857,-156.847,172.829,50.645,160.298
C08895=1018.687,395.611,-156.803,172.818,50.645,160.296
C08896=1018.677,395.366,-156.760,172.807,50.645,160.294
C08897=1018.668,395.119,-156.717,172.796,50.646,160.292
C08898=1018.658,394.873,-156.673,172.784,50.646,160.290
C08899=1018.649,394.627,-156.630,172.773,50.646,160.288
C08900=1018.639,394.381,-156.587,172.763,50.647,160.287
C08901=1018.630,394.135,-156.543,172.752,50.648,160.285
C08902=1018.620,393.890,-156.500,172.741,50.648,160.283
C08903=1018.610,393.643,-156.457,172.729,50.648,160.281
C08904=1018.601,393.397,-156.413,172.718,50.649,160.279
C08905=1018.592,393.151,-156.371,172.707,50.649,160.278
C08906=1018.582,392.905,-156.328,172.696,50.650,160.276
C08907=1018.573,392.659,-156.284,172.686,50.651,160.274
C08908=1018.563,392.413,-156.241,172.675,50.651,160.272
C08909=1018.554,392.167,-156.199,172.664,50.652,160.271
C08910=1018.545,391.920,-156.156,172.653,50.652,160.269
C08911=1018.536,391.675,-156.113,172.643,50.653,160.267
C08912=1018.526,391.428,-156.070,172.631,50.653,160.265
C08913=1018.517,391.182,-156.028,172.620,50.654,160.264
C08914=1018.507,390.937,-155.986,172.610,50.655,160.262
C08915=1018.497,390.690,-155.943,172.599,50.655,160.260
C08916=1018.489,390.444,-155.900,172.588,50.656,160.258
C08917=1018.479,390.198,-155.857,172.578,50.657,160.257
C08918=1018.470,389.952,-155.815,172.567,50.658,160.255
C08919=1018.461,389.706,-155.773,172.556,50.658,160.253
C08920=1018.452,389.460,-155.730,172.546,50.659,160.252
C08921=1018.443,389.213,-155.687,172.536,50.659,160.250
C08922=1018.434,388.967,-155.645,172.525,50.660,160.249
C08923=1018.424,388.721,-155.603,172.515,50.661,160.247
C08924=1018.415,388.475,-155.560,172.504,50.662,160.245
